    |   movel(pose_trans(ref_frame,p[0.137265, 0.127229, -0.000125, -0.013708, 3.141563, 0.000000]),accel_mss,speed_ms,0,0.001)
    |   movel(pose_trans(ref_frame,p[0.137004, 0.127246, -0.000125, -0.013708, 3.141563, 0.000000]),accel_mss,speed_ms,0,0.001)
    |   movel(pose_trans(ref_frame,p[0.136743, 0.127266, -0.000125, -0.013708, 3.141563, 0.000000]),accel_mss,speed_ms,0,0.001)
    |   movel(pose_trans(ref_frame,p[0.136691, 0.127279, -0.000125, -0.013708, 3.141563, -0.000000]),accel_mss,speed_ms,0,0.001)
    |   movel(pose_trans(ref_frame,p[0.136647, 0.127310, -0.000125, -0.013708, 3.141563, -0.000000]),accel_mss,speed_ms,0,0.001)
    |   movel(pose_trans(ref_frame,p[0.136567, 0.127429, -0.000125, -0.013708, 3.141563, -0.000000]),accel_mss,speed_ms,0,0.001)
    |   movel(pose_trans(ref_frame,p[0.136537, 0.127569, -0.000125, -0.013708, 3.141563, -0.000000]),accel_mss,speed_ms,0,0.001)
    |   movel(pose_trans(ref_frame,p[0.136528, 0.128292, -0.000125, -0.013708, 3.141563, -0.000000]),accel_mss,speed_ms,0,0.001)
    |   movel(pose_trans(ref_frame,p[0.136524, 0.129016, -0.000125, -0.013708, 3.141563, -0.000000]),accel_mss,speed_ms,0,0.001)
    |   movel(pose_trans(ref_frame,p[0.136527, 0.129739, -0.000125, -0.013708, 3.141563, 0.000000]),accel_mss,speed_ms,0,0.001)
    |   movel(pose_trans(ref_frame,p[0.136535, 0.130463, -0.000125, -0.013708, 3.141563, 0.000000]),accel_mss,speed_ms,0,0.001)
    |   movel(pose_trans(ref_frame,p[0.136564, 0.130603, -0.000125, -0.013708, 3.141563, 0.000000]),accel_mss,speed_ms,0,0.001)
    |   movel(pose_trans(ref_frame,p[0.136644, 0.130721, -0.000125, -0.013708, 3.141563, 0.000000]),accel_mss,speed_ms,0,0.001)
    |   movel(pose_trans(ref_frame,p[0.136735, 0.130785, -0.000125, -0.013708, 3.141563, 0.000000]),accel_mss,speed_ms,0,0.001)
    |   movel(pose_trans(ref_frame,p[0.136842, 0.130814, -0.000125, -0.013708, 3.141563, -0.000000]),accel_mss,speed_ms,0,0.001)
    |   movel(pose_trans(ref_frame,p[0.137118, 0.130836, -0.000125, -0.013708, 3.141563, 0.000000]),accel_mss,speed_ms,0,0.001)
    |   movel(pose_trans(ref_frame,p[0.137394, 0.130848, -0.000125, -0.013708, 3.141563, 0.000000]),accel_mss,speed_ms,0,0.001)
    |   movel(pose_trans(ref_frame,p[0.137672, 0.130852, -0.000125, -0.013708, 3.141563, -0.000000]),accel_mss,speed_ms,0,0.001)
    |   movel(pose_trans(ref_frame,p[0.137949, 0.130847, -0.000125, -0.013708, 3.141563, -0.000000]),accel_mss,speed_ms,0,0.001)
    |   movel(pose_trans(ref_frame,p[0.138052, 0.130824, -0.000125, -0.013708, 3.141563, 0.000000]),accel_mss,speed_ms,0,0.001)
    |   movel(pose_trans(ref_frame,p[0.138139, 0.130764, -0.000125, -0.013708, 3.141563, -0.000000]),accel_mss,speed_ms,0,0.001)
    |   movel(pose_trans(ref_frame,p[0.138160, 0.130734, -0.000125, -0.013708, 3.141563, 0.000000]),accel_mss,speed_ms,0,0.001)
    |   movel(pose_trans(ref_frame,p[0.138170, 0.130699, -0.000125, -0.013708, 3.141563, 0.000000]),accel_mss,speed_ms,0,0.001)
    |   movel(pose_trans(ref_frame,p[0.138184, 0.130572, -0.000125, -0.013708, 3.141563, 0.000000]),accel_mss,speed_ms,0,0.001)
    |   movel(pose_trans(ref_frame,p[0.138196, 0.130446, -0.000125, -0.013708, 3.141563, 0.000000]),accel_mss,speed_ms,0,0.001)
    |   movel(pose_trans(ref_frame,p[0.138208, 0.130292, -0.000125, -0.013708, 3.141563, 0.000000]),accel_mss,speed_ms,0,0.001)
    |   movel(pose_trans(ref_frame,p[0.138216, 0.130139, -0.000125, -0.013708, 3.141563, -0.000000]),accel_mss,speed_ms,0,0.001)
    |   movel(pose_trans(ref_frame,p[0.138221, 0.129964, -0.000125, -0.013708, 3.141563, 0.000000]),accel_mss,speed_ms,0,0.001)
    |   movel(pose_trans(ref_frame,p[0.138224, 0.129790, -0.000125, -0.013708, 3.141563, 0.000000]),accel_mss,speed_ms,0,0.001)
    |   movel(pose_trans(ref_frame,p[0.138229, 0.128894, -0.000125, -0.013708, 3.141563, -0.000000]),accel_mss,speed_ms,0,0.001)
    |   movel(pose_trans(ref_frame,p[0.139247, 0.128889, -0.000125, -0.013708, 3.141563, 0.000000]),accel_mss,speed_ms,0,0.001)
    |   movel(pose_trans(ref_frame,p[0.139445, 0.128890, -0.000125, -0.013708, 3.141563, 0.000000]),accel_mss,speed_ms,0,0.001)
    |   movel(pose_trans(ref_frame,p[0.139643, 0.128894, -0.000125, -0.013708, 3.141563, -0.000000]),accel_mss,speed_ms,0,0.001)
    |   movel(pose_trans(ref_frame,p[0.139818, 0.128901, -0.000125, -0.013708, 3.141563, 0.000000]),accel_mss,speed_ms,0,0.001)
    |   movel(pose_trans(ref_frame,p[0.139992, 0.128912, -0.000125, -0.013708, 3.141563, -0.000000]),accel_mss,speed_ms,0,0.001)
    |   movel(pose_trans(ref_frame,p[0.140137, 0.128924, -0.000125, -0.013708, 3.141563, 0.000000]),accel_mss,speed_ms,0,0.001)
    |   movel(pose_trans(ref_frame,p[0.140281, 0.128939, -0.000125, -0.013708, 3.141563, -0.000000]),accel_mss,speed_ms,0,0.001)
    |   movel(pose_trans(ref_frame,p[0.140321, 0.128950, -0.000125, -0.013708, 3.141563, 0.000000]),accel_mss,speed_ms,0,0.001)
    |   movel(pose_trans(ref_frame,p[0.140355, 0.128974, -0.000125, -0.013708, 3.141563, -0.000000]),accel_mss,speed_ms,0,0.001)
    |   movel(pose_trans(ref_frame,p[0.140380, 0.129009, -0.000125, -0.013708, 3.141563, 0.000000]),accel_mss,speed_ms,0,0.001)
    |   movel(pose_trans(ref_frame,p[0.140391, 0.129049, -0.000125, -0.013708, 3.141563, 0.000000]),accel_mss,speed_ms,0,0.001)
    |   movel(pose_trans(ref_frame,p[0.140406, 0.129193, -0.000125, -0.013708, 3.141563, 0.000000]),accel_mss,speed_ms,0,0.001)
    |   movel(pose_trans(ref_frame,p[0.140418, 0.129337, -0.000125, -0.013708, 3.141563, -0.000000]),accel_mss,speed_ms,0,0.001)
    |   movel(pose_trans(ref_frame,p[0.140429, 0.129512, -0.000125, -0.013708, 3.141563, 0.000000]),accel_mss,speed_ms,0,0.001)
    |   movel(pose_trans(ref_frame,p[0.140436, 0.129686, -0.000125, -0.013708, 3.141563, 0.000000]),accel_mss,speed_ms,0,0.001)
    |   movel(pose_trans(ref_frame,p[0.140440, 0.129885, -0.000125, -0.013708, 3.141563, 0.000000]),accel_mss,speed_ms,0,0.001)
    |   movel(pose_trans(ref_frame,p[0.140441, 0.130083, -0.000125, -0.013708, 3.141563, -0.000000]),accel_mss,speed_ms,0,0.001)
    |   movel(pose_trans(ref_frame,p[0.140435, 0.131101, -0.000125, -0.013708, 3.141563, 0.000000]),accel_mss,speed_ms,0,0.001)
    |   movel(pose_trans(ref_frame,p[0.139540, 0.131106, -0.000125, -0.013708, 3.141563, -0.000000]),accel_mss,speed_ms,0,0.001)
    |   movel(pose_trans(ref_frame,p[0.139365, 0.131109, -0.000125, -0.013708, 3.141563, 0.000000]),accel_mss,speed_ms,0,0.001)
    |   movel(pose_trans(ref_frame,p[0.139191, 0.131115, -0.000125, -0.013708, 3.141563, 0.000000]),accel_mss,speed_ms,0,0.001)
    |   movel(pose_trans(ref_frame,p[0.139036, 0.131123, -0.000125, -0.013708, 3.141563, 0.000000]),accel_mss,speed_ms,0,0.001)
    |   movel(pose_trans(ref_frame,p[0.138882, 0.131136, -0.000125, -0.013708, 3.141563, -0.000000]),accel_mss,speed_ms,0,0.001)
    |   movel(pose_trans(ref_frame,p[0.138755, 0.131149, -0.000125, -0.013708, 3.141563, -0.000000]),accel_mss,speed_ms,0,0.001)
    |   movel(pose_trans(ref_frame,p[0.138628, 0.131164, -0.000125, -0.013708, 3.141563, 0.000000]),accel_mss,speed_ms,0,0.001)
    |   movel(pose_trans(ref_frame,p[0.138590, 0.131175, -0.000125, -0.013708, 3.141563, 0.000000]),accel_mss,speed_ms,0,0.001)
    |   movel(pose_trans(ref_frame,p[0.138558, 0.131198, -0.000125, -0.013708, 3.141563, -0.000000]),accel_mss,speed_ms,0,0.001)
    |   movel(pose_trans(ref_frame,p[0.138500, 0.131284, -0.000125, -0.013708, 3.141563, -0.000000]),accel_mss,speed_ms,0,0.001)
    |   movel(pose_trans(ref_frame,p[0.138478, 0.131386, -0.000125, -0.013708, 3.141563, 0.000000]),accel_mss,speed_ms,0,0.001)
    |   movel(pose_trans(ref_frame,p[0.138476, 0.131664, -0.000125, -0.013708, 3.141563, 0.000000]),accel_mss,speed_ms,0,0.001)
    |   movel(pose_trans(ref_frame,p[0.138482, 0.131941, -0.000125, -0.013708, 3.141563, 0.000000]),accel_mss,speed_ms,0,0.001)
    |   movel(pose_trans(ref_frame,p[0.138497, 0.132218, -0.000125, -0.013708, 3.141563, -0.000000]),accel_mss,speed_ms,0,0.001)
    |   movel(pose_trans(ref_frame,p[0.138520, 0.132493, -0.000125, -0.013708, 3.141563, 0.000000]),accel_mss,speed_ms,0,0.001)
    |   movel(pose_trans(ref_frame,p[0.138550, 0.132601, -0.000125, -0.013708, 3.141563, -0.000000]),accel_mss,speed_ms,0,0.001)
    |   movel(pose_trans(ref_frame,p[0.138614, 0.132691, -0.000125, -0.013708, 3.141563, 0.000000]),accel_mss,speed_ms,0,0.001)
    |   movel(pose_trans(ref_frame,p[0.138656, 0.132723, -0.000125, -0.013708, 3.141563, -0.000000]),accel_mss,speed_ms,0,0.001)
    |   movel(pose_trans(ref_frame,p[0.138705, 0.132741, -0.000125, -0.013708, 3.141563, 0.000000]),accel_mss,speed_ms,0,0.001)
    |   movel(pose_trans(ref_frame,p[0.138816, 0.132762, -0.000125, -0.013708, 3.141563, 0.000000]),accel_mss,speed_ms,0,0.001)
    |   movel(pose_trans(ref_frame,p[0.138928, 0.132780, -0.000125, -0.013708, 3.141563, -0.000000]),accel_mss,speed_ms,0,0.001)
    |   movel(pose_trans(ref_frame,p[0.139065, 0.132795, -0.000125, -0.013708, 3.141563, -0.000000]),accel_mss,speed_ms,0,0.001)
    |   movel(pose_trans(ref_frame,p[0.139202, 0.132806, -0.000125, -0.013708, 3.141563, -0.000000]),accel_mss,speed_ms,0,0.001)
    |   movel(pose_trans(ref_frame,p[0.139352, 0.132811, -0.000125, -0.013708, 3.141563, 0.000000]),accel_mss,speed_ms,0,0.001)
    |   movel(pose_trans(ref_frame,p[0.139502, 0.132812, -0.000125, -0.013708, 3.141563, 0.000000]),accel_mss,speed_ms,0,0.001)
    |   movel(pose_trans(ref_frame,p[0.139651, 0.132812, -0.000125, -0.013708, 3.141563, 0.000000]),accel_mss,speed_ms,0,0.001)
    |   movel(pose_trans(ref_frame,p[0.139800, 0.132816, -0.000125, -0.013708, 3.141563, -0.000000]),accel_mss,speed_ms,0,0.001)
    |   movel(pose_trans(ref_frame,p[0.139934, 0.132823, -0.000125, -0.013708, 3.141563, 0.000000]),accel_mss,speed_ms,0,0.001)
    |   movel(pose_trans(ref_frame,p[0.140066, 0.132834, -0.000125, -0.013708, 3.141563, -0.000000]),accel_mss,speed_ms,0,0.001)
    |   movel(pose_trans(ref_frame,p[0.140175, 0.132846, -0.000125, -0.013708, 3.141563, 0.000000]),accel_mss,speed_ms,0,0.001)
    |   movel(pose_trans(ref_frame,p[0.140283, 0.132861, -0.000125, -0.013708, 3.141563, -0.000000]),accel_mss,speed_ms,0,0.001)
    |   movel(pose_trans(ref_frame,p[0.140322, 0.132873, -0.000125, -0.013708, 3.141563, 0.000000]),accel_mss,speed_ms,0,0.001)
    |   movel(pose_trans(ref_frame,p[0.140354, 0.132897, -0.000125, -0.013708, 3.141563, 0.000000]),accel_mss,speed_ms,0,0.001)
    |   movel(pose_trans(ref_frame,p[0.140379, 0.132931, -0.000125, -0.013708, 3.141563, -0.000000]),accel_mss,speed_ms,0,0.001)
    |   movel(pose_trans(ref_frame,p[0.140391, 0.132972, -0.000125, -0.013708, 3.141563, 0.000000]),accel_mss,speed_ms,0,0.001)
    |   movel(pose_trans(ref_frame,p[0.140405, 0.133116, -0.000125, -0.013708, 3.141563, -0.000000]),accel_mss,speed_ms,0,0.001)
    |   movel(pose_trans(ref_frame,p[0.140417, 0.133260, -0.000125, -0.013708, 3.141563, -0.000000]),accel_mss,speed_ms,0,0.001)
    |   movel(pose_trans(ref_frame,p[0.140429, 0.133435, -0.000125, -0.013708, 3.141563, -0.000000]),accel_mss,speed_ms,0,0.001)
    |   movel(pose_trans(ref_frame,p[0.140436, 0.133609, -0.000125, -0.013708, 3.141563, -0.000000]),accel_mss,speed_ms,0,0.001)
    |   movel(pose_trans(ref_frame,p[0.140440, 0.133808, -0.000125, -0.013708, 3.141563, 0.000000]),accel_mss,speed_ms,0,0.001)
    |   movel(pose_trans(ref_frame,p[0.140441, 0.134006, -0.000125, -0.013708, 3.141563, -0.000000]),accel_mss,speed_ms,0,0.001)
    |   movel(pose_trans(ref_frame,p[0.140435, 0.135024, -0.000125, -0.013708, 3.141563, 0.000000]),accel_mss,speed_ms,0,0.001)
    |   movel(pose_trans(ref_frame,p[0.139540, 0.135029, -0.000125, -0.013708, 3.141563, 0.000000]),accel_mss,speed_ms,0,0.001)
    |   movel(pose_trans(ref_frame,p[0.139365, 0.135032, -0.000125, -0.013708, 3.141563, 0.000000]),accel_mss,speed_ms,0,0.001)
    |   movel(pose_trans(ref_frame,p[0.139191, 0.135037, -0.000125, -0.013708, 3.141563, -0.000000]),accel_mss,speed_ms,0,0.001)
    |   movel(pose_trans(ref_frame,p[0.139037, 0.135045, -0.000125, -0.013708, 3.141563, -0.000000]),accel_mss,speed_ms,0,0.001)
    |   movel(pose_trans(ref_frame,p[0.138884, 0.135057, -0.000125, -0.013708, 3.141563, -0.000000]),accel_mss,speed_ms,0,0.001)
    |   movel(pose_trans(ref_frame,p[0.138757, 0.135069, -0.000125, -0.013708, 3.141563, 0.000000]),accel_mss,speed_ms,0,0.001)
    |   movel(pose_trans(ref_frame,p[0.138630, 0.135083, -0.000125, -0.013708, 3.141563, -0.000000]),accel_mss,speed_ms,0,0.001)
    |   movel(pose_trans(ref_frame,p[0.138595, 0.135093, -0.000125, -0.013708, 3.141563, 0.000000]),accel_mss,speed_ms,0,0.001)
    |   movel(pose_trans(ref_frame,p[0.138564, 0.135115, -0.000125, -0.013708, 3.141563, 0.000000]),accel_mss,speed_ms,0,0.001)
    |   movel(pose_trans(ref_frame,p[0.138543, 0.135145, -0.000125, -0.013708, 3.141563, 0.000000]),accel_mss,speed_ms,0,0.001)
    |   movel(pose_trans(ref_frame,p[0.138533, 0.135181, -0.000125, -0.013708, 3.141563, 0.000000]),accel_mss,speed_ms,0,0.001)
    |   movel(pose_trans(ref_frame,p[0.138519, 0.135307, -0.000125, -0.013708, 3.141563, 0.000000]),accel_mss,speed_ms,0,0.001)
    |   movel(pose_trans(ref_frame,p[0.138506, 0.135434, -0.000125, -0.013708, 3.141563, 0.000000]),accel_mss,speed_ms,0,0.001)
    |   movel(pose_trans(ref_frame,p[0.138495, 0.135588, -0.000125, -0.013708, 3.141563, 0.000000]),accel_mss,speed_ms,0,0.001)
    |   movel(pose_trans(ref_frame,p[0.138487, 0.135741, -0.000125, -0.013708, 3.141563, 0.000000]),accel_mss,speed_ms,0,0.001)
    |   movel(pose_trans(ref_frame,p[0.138481, 0.135916, -0.000125, -0.013708, 3.141563, 0.000000]),accel_mss,speed_ms,0,0.001)
    |   movel(pose_trans(ref_frame,p[0.138479, 0.136090, -0.000125, -0.013708, 3.141563, 0.000000]),accel_mss,speed_ms,0,0.001)
    |   movel(pose_trans(ref_frame,p[0.138473, 0.136986, -0.000125, -0.013708, 3.141563, -0.000000]),accel_mss,speed_ms,0,0.001)
    |   movel(pose_trans(ref_frame,p[0.137441, 0.136976, -0.000125, -0.013708, 3.141563, 0.000000]),accel_mss,speed_ms,0,0.001)
    |   movel(pose_trans(ref_frame,p[0.137240, 0.136973, -0.000125, -0.013708, 3.141563, 0.000000]),accel_mss,speed_ms,0,0.001)
    |   movel(pose_trans(ref_frame,p[0.137039, 0.136967, -0.000125, -0.013708, 3.141563, 0.000000]),accel_mss,speed_ms,0,0.001)
    |   movel(pose_trans(ref_frame,p[0.136864, 0.136959, -0.000125, -0.013708, 3.141563, 0.000000]),accel_mss,speed_ms,0,0.001)
    |   movel(pose_trans(ref_frame,p[0.136689, 0.136947, -0.000125, -0.013708, 3.141563, 0.000000]),accel_mss,speed_ms,0,0.001)
    |   movel(pose_trans(ref_frame,p[0.136542, 0.136935, -0.000125, -0.013708, 3.141563, 0.000000]),accel_mss,speed_ms,0,0.001)
    |   movel(pose_trans(ref_frame,p[0.136396, 0.136921, -0.000125, -0.013708, 3.141563, 0.000000]),accel_mss,speed_ms,0,0.001)
    |   movel(pose_trans(ref_frame,p[0.136361, 0.136911, -0.000125, -0.013708, 3.141563, 0.000000]),accel_mss,speed_ms,0,0.001)
    |   movel(pose_trans(ref_frame,p[0.136331, 0.136890, -0.000125, -0.013708, 3.141563, 0.000000]),accel_mss,speed_ms,0,0.001)
    |   movel(pose_trans(ref_frame,p[0.136311, 0.136862, -0.000125, -0.013708, 3.141563, -0.000000]),accel_mss,speed_ms,0,0.001)
    |   movel(pose_trans(ref_frame,p[0.136301, 0.136828, -0.000125, -0.013708, 3.141563, -0.000000]),accel_mss,speed_ms,0,0.001)
    |   movel(pose_trans(ref_frame,p[0.136289, 0.136720, -0.000125, -0.013708, 3.141563, -0.000000]),accel_mss,speed_ms,0,0.001)
    |   movel(pose_trans(ref_frame,p[0.136279, 0.136612, -0.000125, -0.013708, 3.141563, -0.000000]),accel_mss,speed_ms,0,0.001)
    |   movel(pose_trans(ref_frame,p[0.136270, 0.136481, -0.000125, -0.013708, 3.141563, -0.000000]),accel_mss,speed_ms,0,0.001)
    |   movel(pose_trans(ref_frame,p[0.136265, 0.136350, -0.000125, -0.013708, 3.141563, -0.000000]),accel_mss,speed_ms,0,0.001)
    |   movel(pose_trans(ref_frame,p[0.136262, 0.136201, -0.000125, -0.013708, 3.141563, -0.000000]),accel_mss,speed_ms,0,0.001)
    |   movel(pose_trans(ref_frame,p[0.136262, 0.136053, -0.000125, -0.013708, 3.141563, -0.000000]),accel_mss,speed_ms,0,0.001)
    |   movel(pose_trans(ref_frame,p[0.136261, 0.135902, -0.000125, -0.013708, 3.141563, -0.000000]),accel_mss,speed_ms,0,0.001)
    |   movel(pose_trans(ref_frame,p[0.136255, 0.135752, -0.000125, -0.013708, 3.141563, 0.000000]),accel_mss,speed_ms,0,0.001)
    |   movel(pose_trans(ref_frame,p[0.136244, 0.135614, -0.000125, -0.013708, 3.141563, -0.000000]),accel_mss,speed_ms,0,0.001)
    |   movel(pose_trans(ref_frame,p[0.136227, 0.135476, -0.000125, -0.013708, 3.141563, 0.000000]),accel_mss,speed_ms,0,0.001)
    |   movel(pose_trans(ref_frame,p[0.136209, 0.135364, -0.000125, -0.013708, 3.141563, 0.000000]),accel_mss,speed_ms,0,0.001)
    |   movel(pose_trans(ref_frame,p[0.136186, 0.135252, -0.000125, -0.013708, 3.141563, 0.000000]),accel_mss,speed_ms,0,0.001)
    |   movel(pose_trans(ref_frame,p[0.136167, 0.135201, -0.000125, -0.013708, 3.141563, -0.000000]),accel_mss,speed_ms,0,0.001)
    |   movel(pose_trans(ref_frame,p[0.136134, 0.135157, -0.000125, -0.013708, 3.141563, -0.000000]),accel_mss,speed_ms,0,0.001)
    |   movel(pose_trans(ref_frame,p[0.136043, 0.135094, -0.000125, -0.013708, 3.141563, 0.000000]),accel_mss,speed_ms,0,0.001)
    |   movel(pose_trans(ref_frame,p[0.135937, 0.135065, -0.000125, -0.013708, 3.141563, -0.000000]),accel_mss,speed_ms,0,0.001)
    |   movel(pose_trans(ref_frame,p[0.135661, 0.135044, -0.000125, -0.013708, 3.141563, -0.000000]),accel_mss,speed_ms,0,0.001)
    |   movel(pose_trans(ref_frame,p[0.135384, 0.135032, -0.000125, -0.013708, 3.141563, -0.000000]),accel_mss,speed_ms,0,0.001)
    |   movel(pose_trans(ref_frame,p[0.135107, 0.135029, -0.000125, -0.013708, 3.141563, 0.000000]),accel_mss,speed_ms,0,0.001)
    |   movel(pose_trans(ref_frame,p[0.134830, 0.135034, -0.000125, -0.013708, 3.141563, 0.000000]),accel_mss,speed_ms,0,0.001)
    |   movel(pose_trans(ref_frame,p[0.134727, 0.135057, -0.000125, -0.013708, 3.141563, -0.000000]),accel_mss,speed_ms,0,0.001)
    |   movel(pose_trans(ref_frame,p[0.134641, 0.135116, -0.000125, -0.013708, 3.141563, 0.000000]),accel_mss,speed_ms,0,0.001)
    |   movel(pose_trans(ref_frame,p[0.134619, 0.135146, -0.000125, -0.013708, 3.141563, -0.000000]),accel_mss,speed_ms,0,0.001)
    |   movel(pose_trans(ref_frame,p[0.134609, 0.135181, -0.000125, -0.013708, 3.141563, -0.000000]),accel_mss,speed_ms,0,0.001)
    |   movel(pose_trans(ref_frame,p[0.134595, 0.135309, -0.000125, -0.013708, 3.141563, 0.000000]),accel_mss,speed_ms,0,0.001)
    |   movel(pose_trans(ref_frame,p[0.134583, 0.135437, -0.000125, -0.013708, 3.141563, 0.000000]),accel_mss,speed_ms,0,0.001)
    |   movel(pose_trans(ref_frame,p[0.134571, 0.135591, -0.000125, -0.013708, 3.141563, 0.000000]),accel_mss,speed_ms,0,0.001)
    |   movel(pose_trans(ref_frame,p[0.134563, 0.135746, -0.000125, -0.013708, 3.141563, -0.000000]),accel_mss,speed_ms,0,0.001)
    |   movel(pose_trans(ref_frame,p[0.134557, 0.135921, -0.000125, -0.013708, 3.141563, 0.000000]),accel_mss,speed_ms,0,0.001)
    |   movel(pose_trans(ref_frame,p[0.134555, 0.136097, -0.000125, -0.013708, 3.141563, -0.000000]),accel_mss,speed_ms,0,0.001)
    |   movel(pose_trans(ref_frame,p[0.134548, 0.136999, -0.000125, -0.013708, 3.141563, 0.000000]),accel_mss,speed_ms,0,0.001)
    |   movel(pose_trans(ref_frame,p[0.133508, 0.136975, -0.000125, -0.013708, 3.141563, 0.000000]),accel_mss,speed_ms,0,0.001)
    |   movel(pose_trans(ref_frame,p[0.133308, 0.136970, -0.000125, -0.013708, 3.141563, -0.000000]),accel_mss,speed_ms,0,0.001)
    |   movel(pose_trans(ref_frame,p[0.133107, 0.136963, -0.000125, -0.013708, 3.141563, 0.000000]),accel_mss,speed_ms,0,0.001)
    |   movel(pose_trans(ref_frame,p[0.132935, 0.136956, -0.000125, -0.013708, 3.141563, 0.000000]),accel_mss,speed_ms,0,0.001)
    |   movel(pose_trans(ref_frame,p[0.132763, 0.136947, -0.000125, -0.013708, 3.141563, -0.000000]),accel_mss,speed_ms,0,0.001)
    |   movel(pose_trans(ref_frame,p[0.132615, 0.136938, -0.000125, -0.013708, 3.141563, -0.000000]),accel_mss,speed_ms,0,0.001)
    |   movel(pose_trans(ref_frame,p[0.132466, 0.136929, -0.000125, -0.013708, 3.141563, 0.000000]),accel_mss,speed_ms,0,0.001)
    |   movel(pose_trans(ref_frame,p[0.132448, 0.136924, -0.000125, -0.013708, 3.141563, -0.000000]),accel_mss,speed_ms,0,0.001)
    |   movel(pose_trans(ref_frame,p[0.132432, 0.136914, -0.000125, -0.013708, 3.141563, -0.000000]),accel_mss,speed_ms,0,0.001)
    |   movel(pose_trans(ref_frame,p[0.132421, 0.136898, -0.000125, -0.013708, 3.141563, 0.000000]),accel_mss,speed_ms,0,0.001)
    |   movel(pose_trans(ref_frame,p[0.132417, 0.136880, -0.000125, -0.013708, 3.141563, -0.000000]),accel_mss,speed_ms,0,0.001)
    |   movel(pose_trans(ref_frame,p[0.132411, 0.136730, -0.000125, -0.013708, 3.141563, -0.000000]),accel_mss,speed_ms,0,0.001)
    |   movel(pose_trans(ref_frame,p[0.132406, 0.136581, -0.000125, -0.013708, 3.141563, 0.000000]),accel_mss,speed_ms,0,0.001)
    |   movel(pose_trans(ref_frame,p[0.132401, 0.136409, -0.000125, -0.013708, 3.141563, -0.000000]),accel_mss,speed_ms,0,0.001)
    |   movel(pose_trans(ref_frame,p[0.132398, 0.136236, -0.000125, -0.013708, 3.141563, 0.000000]),accel_mss,speed_ms,0,0.001)
    |   movel(pose_trans(ref_frame,p[0.132396, 0.136035, -0.000125, -0.013708, 3.141563, -0.000000]),accel_mss,speed_ms,0,0.001)
    |   movel(pose_trans(ref_frame,p[0.132395, 0.135834, -0.000125, -0.013708, 3.141563, -0.000000]),accel_mss,speed_ms,0,0.001)
    |   movel(pose_trans(ref_frame,p[0.132395, 0.134791, -0.000125, -0.013708, 3.141563, 0.000000]),accel_mss,speed_ms,0,0.001)
    |   movel(pose_trans(ref_frame,p[0.133279, 0.134766, -0.000125, -0.013708, 3.141563, 0.000000]),accel_mss,speed_ms,0,0.001)
    |   movel(pose_trans(ref_frame,p[0.133451, 0.134760, -0.000125, -0.013708, 3.141563, 0.000000]),accel_mss,speed_ms,0,0.001)
    |   movel(pose_trans(ref_frame,p[0.133623, 0.134751, -0.000125, -0.013708, 3.141563, 0.000000]),accel_mss,speed_ms,0,0.001)
    |   movel(pose_trans(ref_frame,p[0.133774, 0.134741, -0.000125, -0.013708, 3.141563, 0.000000]),accel_mss,speed_ms,0,0.001)
    |   movel(pose_trans(ref_frame,p[0.133924, 0.134727, -0.000125, -0.013708, 3.141563, 0.000000]),accel_mss,speed_ms,0,0.001)
    |   movel(pose_trans(ref_frame,p[0.134049, 0.134713, -0.000125, -0.013708, 3.141563, 0.000000]),accel_mss,speed_ms,0,0.001)
    |   movel(pose_trans(ref_frame,p[0.134174, 0.134698, -0.000125, -0.013708, 3.141563, 0.000000]),accel_mss,speed_ms,0,0.001)
    |   movel(pose_trans(ref_frame,p[0.134207, 0.134688, -0.000125, -0.013708, 3.141563, -0.000000]),accel_mss,speed_ms,0,0.001)
    |   movel(pose_trans(ref_frame,p[0.134235, 0.134668, -0.000125, -0.013708, 3.141563, 0.000000]),accel_mss,speed_ms,0,0.001)
    |   movel(pose_trans(ref_frame,p[0.134289, 0.134588, -0.000125, -0.013708, 3.141563, -0.000000]),accel_mss,speed_ms,0,0.001)
    |   movel(pose_trans(ref_frame,p[0.134309, 0.134492, -0.000125, -0.013708, 3.141563, -0.000000]),accel_mss,speed_ms,0,0.001)
    |   movel(pose_trans(ref_frame,p[0.134307, 0.134213, -0.000125, -0.013708, 3.141563, 0.000000]),accel_mss,speed_ms,0,0.001)
    |   movel(pose_trans(ref_frame,p[0.134298, 0.133934, -0.000125, -0.013708, 3.141563, 0.000000]),accel_mss,speed_ms,0,0.001)
    |   movel(pose_trans(ref_frame,p[0.134281, 0.133656, -0.000125, -0.013708, 3.141563, 0.000000]),accel_mss,speed_ms,0,0.001)
    |   movel(pose_trans(ref_frame,p[0.134257, 0.133379, -0.000125, -0.013708, 3.141563, -0.000000]),accel_mss,speed_ms,0,0.001)
    |   movel(pose_trans(ref_frame,p[0.134228, 0.133277, -0.000125, -0.013708, 3.141563, -0.000000]),accel_mss,speed_ms,0,0.001)
    |   movel(pose_trans(ref_frame,p[0.134167, 0.133191, -0.000125, -0.013708, 3.141563, -0.000000]),accel_mss,speed_ms,0,0.001)
    |   movel(pose_trans(ref_frame,p[0.134055, 0.133115, -0.000125, -0.013708, 3.141563, 0.000000]),accel_mss,speed_ms,0,0.001)
    |   movel(pose_trans(ref_frame,p[0.133921, 0.133086, -0.000125, -0.013708, 3.141563, -0.000000]),accel_mss,speed_ms,0,0.001)
    |   movel(pose_trans(ref_frame,p[0.133197, 0.133076, -0.000125, -0.013708, 3.141563, -0.000000]),accel_mss,speed_ms,0,0.001)
    |   movel(pose_trans(ref_frame,p[0.132473, 0.133070, -0.000125, -0.013708, 3.141563, 0.000000]),accel_mss,speed_ms,0,0.001)
    |   movel(pose_trans(ref_frame,p[0.131748, 0.133070, -0.000125, -0.013708, 3.141563, 0.000000]),accel_mss,speed_ms,0,0.001)
    |   movel(pose_trans(ref_frame,p[0.131024, 0.133075, -0.000125, -0.013708, 3.141563, 0.000000]),accel_mss,speed_ms,0,0.001)
    |   movel(pose_trans(ref_frame,p[0.130892, 0.133102, -0.000125, -0.013708, 3.141563, -0.000000]),accel_mss,speed_ms,0,0.001)
    |   movel(pose_trans(ref_frame,p[0.130779, 0.133178, -0.000125, -0.013708, 3.141563, 0.000000]),accel_mss,speed_ms,0,0.001)
    |   movel(pose_trans(ref_frame,p[0.130750, 0.133221, -0.000125, -0.013708, 3.141563, 0.000000]),accel_mss,speed_ms,0,0.001)
    |   movel(pose_trans(ref_frame,p[0.130736, 0.133271, -0.000125, -0.013708, 3.141563, 0.000000]),accel_mss,speed_ms,0,0.001)
    |   movel(pose_trans(ref_frame,p[0.130718, 0.133527, -0.000125, -0.013708, 3.141563, 0.000000]),accel_mss,speed_ms,0,0.001)
    |   movel(pose_trans(ref_frame,p[0.130701, 0.133784, -0.000125, -0.013708, 3.141563, 0.000000]),accel_mss,speed_ms,0,0.001)
    |   movel(pose_trans(ref_frame,p[0.130685, 0.134087, -0.000125, -0.013708, 3.141563, -0.000000]),accel_mss,speed_ms,0,0.001)
    |   movel(pose_trans(ref_frame,p[0.130674, 0.134391, -0.000125, -0.013708, 3.141563, -0.000000]),accel_mss,speed_ms,0,0.001)
    |   movel(pose_trans(ref_frame,p[0.130666, 0.134741, -0.000125, -0.013708, 3.141563, 0.000000]),accel_mss,speed_ms,0,0.001)
    |   movel(pose_trans(ref_frame,p[0.130662, 0.135091, -0.000125, -0.013708, 3.141563, 0.000000]),accel_mss,speed_ms,0,0.001)
    |   movel(pose_trans(ref_frame,p[0.130658, 0.135438, -0.000125, -0.013708, 3.141563, -0.000000]),accel_mss,speed_ms,0,0.001)
    |   movel(pose_trans(ref_frame,p[0.130652, 0.135786, -0.000125, -0.013708, 3.141563, 0.000000]),accel_mss,speed_ms,0,0.001)
    |   movel(pose_trans(ref_frame,p[0.130643, 0.136081, -0.000125, -0.013708, 3.141563, -0.000000]),accel_mss,speed_ms,0,0.001)
    |   movel(pose_trans(ref_frame,p[0.130630, 0.136377, -0.000125, -0.013708, 3.141563, -0.000000]),accel_mss,speed_ms,0,0.001)
    |   movel(pose_trans(ref_frame,p[0.130616, 0.136631, -0.000125, -0.013708, 3.141563, -0.000000]),accel_mss,speed_ms,0,0.001)
    |   movel(pose_trans(ref_frame,p[0.130602, 0.136885, -0.000125, -0.013708, 3.141563, 0.000000]),accel_mss,speed_ms,0,0.001)
    |   movel(pose_trans(ref_frame,p[0.130591, 0.136914, -0.000125, -0.013708, 3.141563, 0.000000]),accel_mss,speed_ms,0,0.001)
    |   movel(pose_trans(ref_frame,p[0.130568, 0.136933, -0.000125, -0.013708, 3.141563, 0.000000]),accel_mss,speed_ms,0,0.001)
    |   movel(pose_trans(ref_frame,p[0.130533, 0.136944, -0.000125, -0.013708, 3.141563, 0.000000]),accel_mss,speed_ms,0,0.001)
    |   movel(pose_trans(ref_frame,p[0.130496, 0.136948, -0.000125, -0.013708, 3.141563, -0.000000]),accel_mss,speed_ms,0,0.001)
    |   movel(pose_trans(ref_frame,p[0.115124, 0.136974, -0.000125, -0.013708, 3.141563, -0.000000]),accel_mss,speed_ms,0,0.001)
    |   movel(pose_trans(ref_frame,p[0.106662, 0.136988, -0.000125, -0.013708, 3.141563, 0.000000]),accel_mss,speed_ms,0,0.001)
    |   movel(pose_trans(ref_frame,p[0.098199, 0.136999, -0.000125, -0.013708, 3.141563, 0.000000]),accel_mss,speed_ms,0,0.001)
    |   movel(pose_trans(ref_frame,p[0.088155, 0.137011, -0.000125, -0.013708, 3.141563, 0.000000]),accel_mss,speed_ms,0,0.001)
    |   movel(pose_trans(ref_frame,p[0.078111, 0.137022, -0.000125, -0.013708, 3.141563, -0.000000]),accel_mss,speed_ms,0,0.001)
    |   movel(pose_trans(ref_frame,p[0.025738, 0.137075, -0.000125, -0.013708, 3.141563, 0.000000]),accel_mss,speed_ms,0,0.001)
    |   movel(pose_trans(ref_frame,p[0.025735, 0.135241, -0.000125, -0.013708, 3.141563, -0.000000]),accel_mss,speed_ms,0,0.001)
    |   movel(pose_trans(ref_frame,p[0.025732, 0.134884, -0.000125, -0.013708, 3.141563, -0.000000]),accel_mss,speed_ms,0,0.001)
    |   movel(pose_trans(ref_frame,p[0.025724, 0.134528, -0.000125, -0.013708, 3.141563, 0.000000]),accel_mss,speed_ms,0,0.001)
    |   movel(pose_trans(ref_frame,p[0.025713, 0.134218, -0.000125, -0.013708, 3.141563, 0.000000]),accel_mss,speed_ms,0,0.001)
    |   movel(pose_trans(ref_frame,p[0.025695, 0.133908, -0.000125, -0.013708, 3.141563, -0.000000]),accel_mss,speed_ms,0,0.001)
    |   movel(pose_trans(ref_frame,p[0.025676, 0.133648, -0.000125, -0.013708, 3.141563, 0.000000]),accel_mss,speed_ms,0,0.001)
    |   movel(pose_trans(ref_frame,p[0.025655, 0.133388, -0.000125, -0.013708, 3.141563, 0.000000]),accel_mss,speed_ms,0,0.001)
    |   movel(pose_trans(ref_frame,p[0.025639, 0.133329, -0.000125, -0.013708, 3.141563, 0.000000]),accel_mss,speed_ms,0,0.001)
    |   movel(pose_trans(ref_frame,p[0.025604, 0.133278, -0.000125, -0.013708, 3.141563, -0.000000]),accel_mss,speed_ms,0,0.001)
    |   movel(pose_trans(ref_frame,p[0.025480, 0.133195, -0.000125, -0.013708, 3.141563, -0.000000]),accel_mss,speed_ms,0,0.001)
    |   movel(pose_trans(ref_frame,p[0.025335, 0.133165, -0.000125, -0.013708, 3.141563, -0.000000]),accel_mss,speed_ms,0,0.001)
    |   movel(pose_trans(ref_frame,p[0.024616, 0.133157, -0.000125, -0.013708, 3.141563, -0.000000]),accel_mss,speed_ms,0,0.001)
    |   movel(pose_trans(ref_frame,p[0.023897, 0.133156, -0.000125, -0.013708, 3.141563, -0.000000]),accel_mss,speed_ms,0,0.001)
    |   movel(pose_trans(ref_frame,p[0.023178, 0.133161, -0.000125, -0.013708, 3.141563, 0.000000]),accel_mss,speed_ms,0,0.001)
    |   movel(pose_trans(ref_frame,p[0.022459, 0.133172, -0.000125, -0.013708, 3.141563, 0.000000]),accel_mss,speed_ms,0,0.001)
    |   movel(pose_trans(ref_frame,p[0.022313, 0.133204, -0.000125, -0.013708, 3.141563, -0.000000]),accel_mss,speed_ms,0,0.001)
    |   movel(pose_trans(ref_frame,p[0.022189, 0.133287, -0.000125, -0.013708, 3.141563, -0.000000]),accel_mss,speed_ms,0,0.001)
    |   movel(pose_trans(ref_frame,p[0.022117, 0.133391, -0.000125, -0.013708, 3.141563, 0.000000]),accel_mss,speed_ms,0,0.001)
    |   movel(pose_trans(ref_frame,p[0.022084, 0.133512, -0.000125, -0.013708, 3.141563, 0.000000]),accel_mss,speed_ms,0,0.001)
    |   movel(pose_trans(ref_frame,p[0.022070, 0.133748, -0.000125, -0.013708, 3.141563, 0.000000]),accel_mss,speed_ms,0,0.001)
    |   movel(pose_trans(ref_frame,p[0.022071, 0.133983, -0.000125, -0.013708, 3.141563, -0.000000]),accel_mss,speed_ms,0,0.001)
    |   movel(pose_trans(ref_frame,p[0.022087, 0.134220, -0.000125, -0.013708, 3.141563, 0.000000]),accel_mss,speed_ms,0,0.001)
    |   movel(pose_trans(ref_frame,p[0.022119, 0.134454, -0.000125, -0.013708, 3.141563, 0.000000]),accel_mss,speed_ms,0,0.001)
    |   movel(pose_trans(ref_frame,p[0.022160, 0.134581, -0.000125, -0.013708, 3.141563, -0.000000]),accel_mss,speed_ms,0,0.001)
    |   movel(pose_trans(ref_frame,p[0.022239, 0.134690, -0.000125, -0.013708, 3.141563, 0.000000]),accel_mss,speed_ms,0,0.001)
    |   movel(pose_trans(ref_frame,p[0.022291, 0.134729, -0.000125, -0.013708, 3.141563, 0.000000]),accel_mss,speed_ms,0,0.001)
    |   movel(pose_trans(ref_frame,p[0.022350, 0.134754, -0.000125, -0.013708, 3.141563, 0.000000]),accel_mss,speed_ms,0,0.001)
    |   movel(pose_trans(ref_frame,p[0.022471, 0.134783, -0.000125, -0.013708, 3.141563, -0.000000]),accel_mss,speed_ms,0,0.001)
    |   movel(pose_trans(ref_frame,p[0.022593, 0.134807, -0.000125, -0.013708, 3.141563, 0.000000]),accel_mss,speed_ms,0,0.001)
    |   movel(pose_trans(ref_frame,p[0.022741, 0.134829, -0.000125, -0.013708, 3.141563, 0.000000]),accel_mss,speed_ms,0,0.001)
    |   movel(pose_trans(ref_frame,p[0.022891, 0.134845, -0.000125, -0.013708, 3.141563, 0.000000]),accel_mss,speed_ms,0,0.001)
    |   movel(pose_trans(ref_frame,p[0.023052, 0.134855, -0.000125, -0.013708, 3.141563, 0.000000]),accel_mss,speed_ms,0,0.001)
    |   movel(pose_trans(ref_frame,p[0.023213, 0.134859, -0.000125, -0.013708, 3.141563, 0.000000]),accel_mss,speed_ms,0,0.001)
    |   movel(pose_trans(ref_frame,p[0.024024, 0.134865, -0.000125, -0.013708, 3.141563, 0.000000]),accel_mss,speed_ms,0,0.001)
    |   movel(pose_trans(ref_frame,p[0.024029, 0.135970, -0.000125, -0.013708, 3.141563, 0.000000]),accel_mss,speed_ms,0,0.001)
    |   movel(pose_trans(ref_frame,p[0.024034, 0.137075, -0.000125, -0.013708, 3.141563, -0.000000]),accel_mss,speed_ms,0,0.001)
    |   movel(pose_trans(ref_frame,p[0.022932, 0.137075, -0.000125, -0.013708, 3.141563, 0.000000]),accel_mss,speed_ms,0,0.001)
    |   movel(pose_trans(ref_frame,p[0.021829, 0.137075, -0.000125, -0.013708, 3.141563, 0.000000]),accel_mss,speed_ms,0,0.001)
    |   movel(pose_trans(ref_frame,p[0.021877, 0.136331, -0.000125, -0.013708, 3.141563, 0.000000]),accel_mss,speed_ms,0,0.001)
    |   movel(pose_trans(ref_frame,p[0.021890, 0.135997, -0.000125, -0.013708, 3.141563, -0.000000]),accel_mss,speed_ms,0,0.001)
    |   movel(pose_trans(ref_frame,p[0.021886, 0.135664, -0.000125, -0.013708, 3.141563, -0.000000]),accel_mss,speed_ms,0,0.001)
    |   movel(pose_trans(ref_frame,p[0.021855, 0.135492, -0.000125, -0.013708, 3.141563, 0.000000]),accel_mss,speed_ms,0,0.001)
    |   movel(pose_trans(ref_frame,p[0.021777, 0.135336, -0.000125, -0.013708, 3.141563, -0.000000]),accel_mss,speed_ms,0,0.001)
    |   movel(pose_trans(ref_frame,p[0.021666, 0.135228, -0.000125, -0.013708, 3.141563, -0.000000]),accel_mss,speed_ms,0,0.001)
    |   movel(pose_trans(ref_frame,p[0.021524, 0.135169, -0.000125, -0.013708, 3.141563, -0.000000]),accel_mss,speed_ms,0,0.001)
    |   movel(pose_trans(ref_frame,p[0.021277, 0.135130, -0.000125, -0.013708, 3.141563, -0.000000]),accel_mss,speed_ms,0,0.001)
    |   movel(pose_trans(ref_frame,p[0.021026, 0.135115, -0.000125, -0.013708, 3.141563, -0.000000]),accel_mss,speed_ms,0,0.001)
    |   movel(pose_trans(ref_frame,p[0.020896, 0.135115, -0.000125, -0.013708, 3.141563, 0.000000]),accel_mss,speed_ms,0,0.001)
    |   movel(pose_trans(ref_frame,p[0.020766, 0.135121, -0.000125, -0.013708, 3.141563, 0.000000]),accel_mss,speed_ms,0,0.001)
    |   movel(pose_trans(ref_frame,p[0.020646, 0.135130, -0.000125, -0.013708, 3.141563, 0.000000]),accel_mss,speed_ms,0,0.001)
    |   movel(pose_trans(ref_frame,p[0.020527, 0.135145, -0.000125, -0.013708, 3.141563, 0.000000]),accel_mss,speed_ms,0,0.001)
    |   movel(pose_trans(ref_frame,p[0.020430, 0.135161, -0.000125, -0.013708, 3.141563, 0.000000]),accel_mss,speed_ms,0,0.001)
    |   movel(pose_trans(ref_frame,p[0.020333, 0.135181, -0.000125, -0.013708, 3.141563, 0.000000]),accel_mss,speed_ms,0,0.001)
    |   movel(pose_trans(ref_frame,p[0.020288, 0.135199, -0.000125, -0.013708, 3.141563, 0.000000]),accel_mss,speed_ms,0,0.001)
    |   movel(pose_trans(ref_frame,p[0.020249, 0.135228, -0.000125, -0.013708, 3.141563, 0.000000]),accel_mss,speed_ms,0,0.001)
    |   movel(pose_trans(ref_frame,p[0.020218, 0.135270, -0.000125, -0.013708, 3.141563, 0.000000]),accel_mss,speed_ms,0,0.001)
    |   movel(pose_trans(ref_frame,p[0.020202, 0.135319, -0.000125, -0.013708, 3.141563, 0.000000]),accel_mss,speed_ms,0,0.001)
    |   movel(pose_trans(ref_frame,p[0.020183, 0.135442, -0.000125, -0.013708, 3.141563, 0.000000]),accel_mss,speed_ms,0,0.001)
    |   movel(pose_trans(ref_frame,p[0.020167, 0.135567, -0.000125, -0.013708, 3.141563, 0.000000]),accel_mss,speed_ms,0,0.001)
    |   movel(pose_trans(ref_frame,p[0.020153, 0.135719, -0.000125, -0.013708, 3.141563, -0.000000]),accel_mss,speed_ms,0,0.001)
    |   movel(pose_trans(ref_frame,p[0.020145, 0.135872, -0.000125, -0.013708, 3.141563, -0.000000]),accel_mss,speed_ms,0,0.001)
    |   movel(pose_trans(ref_frame,p[0.020141, 0.136041, -0.000125, -0.013708, 3.141563, -0.000000]),accel_mss,speed_ms,0,0.001)
    |   movel(pose_trans(ref_frame,p[0.020141, 0.136210, -0.000125, -0.013708, 3.141563, -0.000000]),accel_mss,speed_ms,0,0.001)
    |   movel(pose_trans(ref_frame,p[0.020155, 0.137072, -0.000125, -0.013708, 3.141563, 0.000000]),accel_mss,speed_ms,0,0.001)
    |   movel(pose_trans(ref_frame,p[0.019067, 0.137076, -0.000125, -0.013708, 3.141563, 0.000000]),accel_mss,speed_ms,0,0.001)
    |   movel(pose_trans(ref_frame,p[0.017979, 0.137081, -0.000125, -0.013708, 3.141563, 0.000000]),accel_mss,speed_ms,0,0.001)
    |   movel(pose_trans(ref_frame,p[0.017974, 0.136223, -0.000125, -0.013708, 3.141563, -0.000000]),accel_mss,speed_ms,0,0.001)
    |   movel(pose_trans(ref_frame,p[0.017971, 0.136054, -0.000125, -0.013708, 3.141563, -0.000000]),accel_mss,speed_ms,0,0.001)
    |   movel(pose_trans(ref_frame,p[0.017963, 0.135886, -0.000125, -0.013708, 3.141563, 0.000000]),accel_mss,speed_ms,0,0.001)
    |   movel(pose_trans(ref_frame,p[0.017951, 0.135733, -0.000125, -0.013708, 3.141563, 0.000000]),accel_mss,speed_ms,0,0.001)
    |   movel(pose_trans(ref_frame,p[0.017934, 0.135581, -0.000125, -0.013708, 3.141563, -0.000000]),accel_mss,speed_ms,0,0.001)
    |   movel(pose_trans(ref_frame,p[0.017916, 0.135457, -0.000125, -0.013708, 3.141563, 0.000000]),accel_mss,speed_ms,0,0.001)
    |   movel(pose_trans(ref_frame,p[0.017894, 0.135334, -0.000125, -0.013708, 3.141563, 0.000000]),accel_mss,speed_ms,0,0.001)
    |   movel(pose_trans(ref_frame,p[0.017877, 0.135285, -0.000125, -0.013708, 3.141563, 0.000000]),accel_mss,speed_ms,0,0.001)
    |   movel(pose_trans(ref_frame,p[0.017846, 0.135243, -0.000125, -0.013708, 3.141563, -0.000000]),accel_mss,speed_ms,0,0.001)
    |   movel(pose_trans(ref_frame,p[0.017804, 0.135212, -0.000125, -0.013708, 3.141563, -0.000000]),accel_mss,speed_ms,0,0.001)
    |   movel(pose_trans(ref_frame,p[0.017755, 0.135194, -0.000125, -0.013708, 3.141563, 0.000000]),accel_mss,speed_ms,0,0.001)
    |   movel(pose_trans(ref_frame,p[0.017631, 0.135173, -0.000125, -0.013708, 3.141563, -0.000000]),accel_mss,speed_ms,0,0.001)
    |   movel(pose_trans(ref_frame,p[0.017507, 0.135155, -0.000125, -0.013708, 3.141563, 0.000000]),accel_mss,speed_ms,0,0.001)
    |   movel(pose_trans(ref_frame,p[0.017355, 0.135138, -0.000125, -0.013708, 3.141563, 0.000000]),accel_mss,speed_ms,0,0.001)
    |   movel(pose_trans(ref_frame,p[0.017203, 0.135126, -0.000125, -0.013708, 3.141563, -0.000000]),accel_mss,speed_ms,0,0.001)
    |   movel(pose_trans(ref_frame,p[0.017034, 0.135118, -0.000125, -0.013708, 3.141563, 0.000000]),accel_mss,speed_ms,0,0.001)
    |   movel(pose_trans(ref_frame,p[0.016865, 0.135115, -0.000125, -0.013708, 3.141563, -0.000000]),accel_mss,speed_ms,0,0.001)
    |   movel(pose_trans(ref_frame,p[0.016008, 0.135109, -0.000125, -0.013708, 3.141563, -0.000000]),accel_mss,speed_ms,0,0.001)
    |   movel(pose_trans(ref_frame,p[0.016011, 0.134006, -0.000125, -0.013708, 3.141563, -0.000000]),accel_mss,speed_ms,0,0) # end trace
    |   speed_ms    = 1.000
    |   movel(pose_trans(ref_frame,p[0.016011, 0.134006, 0.005000, -0.013708, 3.141563, -0.000000]),accel_mss,speed_ms,0,0.001)
    |   movel(pose_trans(ref_frame,p[0.000000, 0.000000, 0.005000, -0.013708, 3.141563, 0.000000]),accel_mss,speed_ms,0,0.001)
    |   movel(pose_trans(ref_frame,p[0.000000, 0.000000, 0.055000, -0.013708, 3.141563, -0.000000]),accel_mss,speed_ms,0,0.001)
    |   # End of main program
    | end
    | 
    | output_middle()
  Script file /programs/usbdisk/output_RSettings.script
    | def output_RSettings():
    |   # Global parameters:
    |   global speed_ms    = 0.250
    |   global speed_rads  = 0.750
    |   global accel_mss   = 1.200
    |   global accel_radss = 1.200
    |   global blend_radius_m = 0.001
    |   global ref_frame = p[0,0,0,0,0,0]
    | 
    |   #
    |   # TO REMOVE HEADER:
    |   # Go to "Program" -> "Post-Processor Editor"
    |   # Select "Universal Robots"
    |   # Set "INCLUDE_HEADER" to "False"
    |   #
    |   #--------------------------
    |   # Add any default subprograms here
    |   # For example, to drive a gripper as a program call:
    |   # def Gripper_Open():
    |   #   ...
    |   # end
    |   #
    |   # Example to drive a spray gun:
    |   def SprayOn(value):
    |     # use the value as an output:
    |     DO_SPRAY = 5
    |     if value == 0:
    |       set_standard_digital_out(DO_SPRAY, False)
    |     else:
    |       set_standard_digital_out(DO_SPRAY, True)
    |     end
    |   end
    | 
    |   # Example to drive an extruder:
    |   def Extruder(value):
    |     # use the value as an output:
    |     if value < 0:
    |       # stop extruder
    |     else:
    |       # start extruder
    |     end
    |   end
    | 
    |   # Example to move an external axis
    |   def MoveAxis(value):
    |     # use the value as an output:
    |     DO_AXIS_1 = 1
    |     DI_AXIS_1 = 1
    |     if value <= 0:
    |       set_standard_digital_out(DO_AXIS_1, False)
    | 
    |       # Wait for digital input to change state
    |       #while (get_standard_digital_in(DI_AXIS_1) != False):
    |       #  sync()
    |       #end
    |     else:
    |       set_standard_digital_out(DO_AXIS_1, True)
    | 
    |       # Wait for digital input to change state
    |       #while (get_standard_digital_in(DI_AXIS_1) != True):
    |       #  sync()
    |       #end
    |     end
    |   end
    |   #--------------------------
    | 
    | 
    |   # Main program:
    |   # Program generated by RoboDK v5.7.4 for UR10e on 08/01/2025 21:21:43
    |   # Using nominal kinematics.
    |   blend_radius_m = 0.001
    |   speed_ms    = 1.000
    |   ref_frame = p[0.326125, 0.122767, 0.009000, 0.000000, 0.000000, -0.008727]
    |   set_tcp(p[0.000000, 0.000000, 0.252000, 0.000000, 0.000000, 0.000000])
    |   # Show Tool
    |   movej([0.854487, -1.303262, -2.473446, -0.935678, 1.570796, 2.425275],accel_radss,speed_rads,0,0)
    |   movel(pose_trans(ref_frame,p[0.078892, 0.078720, 0.005000, -0.013708, 3.141563, 0.000000]),accel_mss,speed_ms,0,0) # end trace
    |   speed_ms    = 0.002
    |   movel(pose_trans(ref_frame,p[0.078892, 0.078720, -0.000125, -0.013708, 3.141563, -0.000000]),accel_mss,speed_ms,0,0) # end trace
    |   speed_ms    = 0.007
    |   movel(pose_trans(ref_frame,p[0.079868, 0.078932, -0.000125, -0.013708, 3.141563, 0.000000]),accel_mss,speed_ms,0,0.001)
    |   movel(pose_trans(ref_frame,p[0.080833, 0.079163, -0.000125, -0.013708, 3.141563, 0.000000]),accel_mss,speed_ms,0,0.001)
    |   movel(pose_trans(ref_frame,p[0.081602, 0.079416, -0.000125, -0.013708, 3.141563, -0.000000]),accel_mss,speed_ms,0,0.001)
    |   movel(pose_trans(ref_frame,p[0.082359, 0.079687, -0.000125, -0.013708, 3.141563, -0.000000]),accel_mss,speed_ms,0,0.001)
    |   movel(pose_trans(ref_frame,p[0.086688, 0.081714, -0.000125, -0.013708, 3.141563, 0.000000]),accel_mss,speed_ms,0,0.001)
    |   movel(pose_trans(ref_frame,p[0.090570, 0.084347, -0.000125, -0.013708, 3.141563, 0.000000]),accel_mss,speed_ms,0,0.001)
    |   movel(pose_trans(ref_frame,p[0.091420, 0.085053, -0.000125, -0.013708, 3.141563, 0.000000]),accel_mss,speed_ms,0,0.001)
    |   movel(pose_trans(ref_frame,p[0.092243, 0.085789, -0.000125, -0.013708, 3.141563, -0.000000]),accel_mss,speed_ms,0,0.001)
    |   movel(pose_trans(ref_frame,p[0.092902, 0.086419, -0.000125, -0.013708, 3.141563, 0.000000]),accel_mss,speed_ms,0,0.001)
    |   movel(pose_trans(ref_frame,p[0.093542, 0.087070, -0.000125, -0.013708, 3.141563, 0.000000]),accel_mss,speed_ms,0,0.001)
    |   movel(pose_trans(ref_frame,p[0.093889, 0.087440, -0.000125, -0.013708, 3.141563, 0.000000]),accel_mss,speed_ms,0,0.001)
    |   movel(pose_trans(ref_frame,p[0.094230, 0.087815, -0.000125, -0.013708, 3.141563, 0.000000]),accel_mss,speed_ms,0,0.001)
    |   movel(pose_trans(ref_frame,p[0.094772, 0.088440, -0.000125, -0.013708, 3.141563, 0.000000]),accel_mss,speed_ms,0,0.001)
    |   movel(pose_trans(ref_frame,p[0.095297, 0.089081, -0.000125, -0.013708, 3.141563, -0.000000]),accel_mss,speed_ms,0,0.001)
    |   movel(pose_trans(ref_frame,p[0.095678, 0.089569, -0.000125, -0.013708, 3.141563, 0.000000]),accel_mss,speed_ms,0,0.001)
    |   movel(pose_trans(ref_frame,p[0.096049, 0.090066, -0.000125, -0.013708, 3.141563, 0.000000]),accel_mss,speed_ms,0,0.001)
    |   movel(pose_trans(ref_frame,p[0.097201, 0.091759, -0.000125, -0.013708, 3.141563, -0.000000]),accel_mss,speed_ms,0,0.001)
    |   movel(pose_trans(ref_frame,p[0.098242, 0.093541, -0.000125, -0.013708, 3.141563, -0.000000]),accel_mss,speed_ms,0,0.001)
    |   movel(pose_trans(ref_frame,p[0.098866, 0.094765, -0.000125, -0.013708, 3.141563, 0.000000]),accel_mss,speed_ms,0,0.001)
    |   movel(pose_trans(ref_frame,p[0.099437, 0.096026, -0.000125, -0.013708, 3.141563, 0.000000]),accel_mss,speed_ms,0,0.001)
    |   movel(pose_trans(ref_frame,p[0.100019, 0.097672, -0.000125, -0.013708, 3.141563, 0.000000]),accel_mss,speed_ms,0,0.001)
    |   movel(pose_trans(ref_frame,p[0.100523, 0.099369, -0.000125, -0.013708, 3.141563, 0.000000]),accel_mss,speed_ms,0,0) # end trace
    |   speed_ms    = 1.000
    |   movel(pose_trans(ref_frame,p[0.100523, 0.099369, 0.005000, -0.013708, 3.141563, 0.000000]),accel_mss,speed_ms,0,0.001)
    |   movel(pose_trans(ref_frame,p[0.087112, 0.102660, 0.005000, -0.013708, 3.141563, -0.000000]),accel_mss,speed_ms,0,0) # end trace
    |   speed_ms    = 0.002
    |   movel(pose_trans(ref_frame,p[0.087112, 0.102660, -0.000125, -0.013708, 3.141563, -0.000000]),accel_mss,speed_ms,0,0) # end trace
    |   speed_ms    = 0.007
    |   movel(pose_trans(ref_frame,p[0.087463, 0.102752, -0.000125, -0.013708, 3.141563, -0.000000]),accel_mss,speed_ms,0,0.001)
    |   movel(pose_trans(ref_frame,p[0.087821, 0.102816, -0.000125, -0.013708, 3.141563, 0.000000]),accel_mss,speed_ms,0,0.001)
    |   movel(pose_trans(ref_frame,p[0.088167, 0.102847, -0.000125, -0.013708, 3.141563, 0.000000]),accel_mss,speed_ms,0,0.001)
    |   movel(pose_trans(ref_frame,p[0.088514, 0.102847, -0.000125, -0.013708, 3.141563, 0.000000]),accel_mss,speed_ms,0,0.001)
    |   movel(pose_trans(ref_frame,p[0.088877, 0.102814, -0.000125, -0.013708, 3.141563, 0.000000]),accel_mss,speed_ms,0,0.001)
    |   movel(pose_trans(ref_frame,p[0.089235, 0.102751, -0.000125, -0.013708, 3.141563, 0.000000]),accel_mss,speed_ms,0,0.001)
    |   movel(pose_trans(ref_frame,p[0.089634, 0.102650, -0.000125, -0.013708, 3.141563, 0.000000]),accel_mss,speed_ms,0,0.001)
    |   movel(pose_trans(ref_frame,p[0.090026, 0.102526, -0.000125, -0.013708, 3.141563, -0.000000]),accel_mss,speed_ms,0,0.001)
    |   movel(pose_trans(ref_frame,p[0.090266, 0.102437, -0.000125, -0.013708, 3.141563, -0.000000]),accel_mss,speed_ms,0,0.001)
    |   movel(pose_trans(ref_frame,p[0.090502, 0.102340, -0.000125, -0.013708, 3.141563, -0.000000]),accel_mss,speed_ms,0,0.001)
    |   movel(pose_trans(ref_frame,p[0.090671, 0.102259, -0.000125, -0.013708, 3.141563, 0.000000]),accel_mss,speed_ms,0,0.001)
    |   movel(pose_trans(ref_frame,p[0.090831, 0.102163, -0.000125, -0.013708, 3.141563, 0.000000]),accel_mss,speed_ms,0,0.001)
    |   movel(pose_trans(ref_frame,p[0.090992, 0.102049, -0.000125, -0.013708, 3.141563, 0.000000]),accel_mss,speed_ms,0,0.001)
    |   movel(pose_trans(ref_frame,p[0.091143, 0.101922, -0.000125, -0.013708, 3.141563, 0.000000]),accel_mss,speed_ms,0,0.001)
    |   movel(pose_trans(ref_frame,p[0.091360, 0.101720, -0.000125, -0.013708, 3.141563, -0.000000]),accel_mss,speed_ms,0,0.001)
    |   movel(pose_trans(ref_frame,p[0.091572, 0.101513, -0.000125, -0.013708, 3.141563, 0.000000]),accel_mss,speed_ms,0,0.001)
    |   movel(pose_trans(ref_frame,p[0.091779, 0.101301, -0.000125, -0.013708, 3.141563, 0.000000]),accel_mss,speed_ms,0,0.001)
    |   movel(pose_trans(ref_frame,p[0.091981, 0.101085, -0.000125, -0.013708, 3.141563, 0.000000]),accel_mss,speed_ms,0,0.001)
    |   movel(pose_trans(ref_frame,p[0.092104, 0.100938, -0.000125, -0.013708, 3.141563, 0.000000]),accel_mss,speed_ms,0,0.001)
    |   movel(pose_trans(ref_frame,p[0.092216, 0.100781, -0.000125, -0.013708, 3.141563, 0.000000]),accel_mss,speed_ms,0,0.001)
    |   movel(pose_trans(ref_frame,p[0.092307, 0.100629, -0.000125, -0.013708, 3.141563, 0.000000]),accel_mss,speed_ms,0,0.001)
    |   movel(pose_trans(ref_frame,p[0.092383, 0.100468, -0.000125, -0.013708, 3.141563, 0.000000]),accel_mss,speed_ms,0,0.001)
    |   movel(pose_trans(ref_frame,p[0.092470, 0.100248, -0.000125, -0.013708, 3.141563, -0.000000]),accel_mss,speed_ms,0,0.001)
    |   movel(pose_trans(ref_frame,p[0.092549, 0.100024, -0.000125, -0.013708, 3.141563, 0.000000]),accel_mss,speed_ms,0,0.001)
    |   movel(pose_trans(ref_frame,p[0.092669, 0.099587, -0.000125, -0.013708, 3.141563, -0.000000]),accel_mss,speed_ms,0,0.001)
    |   movel(pose_trans(ref_frame,p[0.092743, 0.099139, -0.000125, -0.013708, 3.141563, 0.000000]),accel_mss,speed_ms,0,0.001)
    |   movel(pose_trans(ref_frame,p[0.092785, 0.098610, -0.000125, -0.013708, 3.141563, 0.000000]),accel_mss,speed_ms,0,0.001)
    |   movel(pose_trans(ref_frame,p[0.092793, 0.098080, -0.000125, -0.013708, 3.141563, -0.000000]),accel_mss,speed_ms,0,0.001)
    |   movel(pose_trans(ref_frame,p[0.092765, 0.097519, -0.000125, -0.013708, 3.141563, 0.000000]),accel_mss,speed_ms,0,0.001)
    |   movel(pose_trans(ref_frame,p[0.092703, 0.096961, -0.000125, -0.013708, 3.141563, 0.000000]),accel_mss,speed_ms,0,0.001)
    |   movel(pose_trans(ref_frame,p[0.092608, 0.096423, -0.000125, -0.013708, 3.141563, -0.000000]),accel_mss,speed_ms,0,0.001)
    |   movel(pose_trans(ref_frame,p[0.092476, 0.095893, -0.000125, -0.013708, 3.141563, -0.000000]),accel_mss,speed_ms,0,0.001)
    |   movel(pose_trans(ref_frame,p[0.092409, 0.095667, -0.000125, -0.013708, 3.141563, 0.000000]),accel_mss,speed_ms,0,0.001)
    |   movel(pose_trans(ref_frame,p[0.092337, 0.095443, -0.000125, -0.013708, 3.141563, 0.000000]),accel_mss,speed_ms,0,0.001)
    |   movel(pose_trans(ref_frame,p[0.092262, 0.095233, -0.000125, -0.013708, 3.141563, 0.000000]),accel_mss,speed_ms,0,0.001)
    |   movel(pose_trans(ref_frame,p[0.092182, 0.095026, -0.000125, -0.013708, 3.141563, 0.000000]),accel_mss,speed_ms,0,0.001)
    |   movel(pose_trans(ref_frame,p[0.092110, 0.094854, -0.000125, -0.013708, 3.141563, -0.000000]),accel_mss,speed_ms,0,0.001)
    |   movel(pose_trans(ref_frame,p[0.092033, 0.094685, -0.000125, -0.013708, 3.141563, -0.000000]),accel_mss,speed_ms,0,0.001)
    |   movel(pose_trans(ref_frame,p[0.091986, 0.094604, -0.000125, -0.013708, 3.141563, 0.000000]),accel_mss,speed_ms,0,0.001)
    |   movel(pose_trans(ref_frame,p[0.091926, 0.094532, -0.000125, -0.013708, 3.141563, -0.000000]),accel_mss,speed_ms,0,0.001)
    |   movel(pose_trans(ref_frame,p[0.091668, 0.094355, -0.000125, -0.013708, 3.141563, 0.000000]),accel_mss,speed_ms,0,0.001)
    |   movel(pose_trans(ref_frame,p[0.091363, 0.094284, -0.000125, -0.013708, 3.141563, 0.000000]),accel_mss,speed_ms,0,0.001)
    |   movel(pose_trans(ref_frame,p[0.090817, 0.094283, -0.000125, -0.013708, 3.141563, 0.000000]),accel_mss,speed_ms,0,0.001)
    |   movel(pose_trans(ref_frame,p[0.090272, 0.094324, -0.000125, -0.013708, 3.141563, 0.000000]),accel_mss,speed_ms,0,0.001)
    |   movel(pose_trans(ref_frame,p[0.089634, 0.094424, -0.000125, -0.013708, 3.141563, 0.000000]),accel_mss,speed_ms,0,0.001)
    |   movel(pose_trans(ref_frame,p[0.089006, 0.094572, -0.000125, -0.013708, 3.141563, -0.000000]),accel_mss,speed_ms,0,0.001)
    |   movel(pose_trans(ref_frame,p[0.088394, 0.094768, -0.000125, -0.013708, 3.141563, 0.000000]),accel_mss,speed_ms,0,0.001)
    |   movel(pose_trans(ref_frame,p[0.087800, 0.095012, -0.000125, -0.013708, 3.141563, 0.000000]),accel_mss,speed_ms,0,0.001)
    |   movel(pose_trans(ref_frame,p[0.087450, 0.095185, -0.000125, -0.013708, 3.141563, -0.000000]),accel_mss,speed_ms,0,0.001)
    |   movel(pose_trans(ref_frame,p[0.087113, 0.095382, -0.000125, -0.013708, 3.141563, 0.000000]),accel_mss,speed_ms,0,0.001)
    |   movel(pose_trans(ref_frame,p[0.086733, 0.095631, -0.000125, -0.013708, 3.141563, 0.000000]),accel_mss,speed_ms,0,0.001)
    |   movel(pose_trans(ref_frame,p[0.086364, 0.095897, -0.000125, -0.013708, 3.141563, -0.000000]),accel_mss,speed_ms,0,0.001)
    |   movel(pose_trans(ref_frame,p[0.086019, 0.096167, -0.000125, -0.013708, 3.141563, 0.000000]),accel_mss,speed_ms,0,0.001)
    |   movel(pose_trans(ref_frame,p[0.085686, 0.096452, -0.000125, -0.013708, 3.141563, 0.000000]),accel_mss,speed_ms,0,0.001)
    |   movel(pose_trans(ref_frame,p[0.085448, 0.096684, -0.000125, -0.013708, 3.141563, -0.000000]),accel_mss,speed_ms,0,0.001)
    |   movel(pose_trans(ref_frame,p[0.085234, 0.096938, -0.000125, -0.013708, 3.141563, 0.000000]),accel_mss,speed_ms,0,0.001)
    |   movel(pose_trans(ref_frame,p[0.084848, 0.097539, -0.000125, -0.013708, 3.141563, -0.000000]),accel_mss,speed_ms,0,0.001)
    |   movel(pose_trans(ref_frame,p[0.084569, 0.098197, -0.000125, -0.013708, 3.141563, -0.000000]),accel_mss,speed_ms,0,0.001)
    |   movel(pose_trans(ref_frame,p[0.084427, 0.098849, -0.000125, -0.013708, 3.141563, -0.000000]),accel_mss,speed_ms,0,0.001)
    |   movel(pose_trans(ref_frame,p[0.084421, 0.099516, -0.000125, -0.013708, 3.141563, -0.000000]),accel_mss,speed_ms,0,0.001)
    |   movel(pose_trans(ref_frame,p[0.084552, 0.100168, -0.000125, -0.013708, 3.141563, -0.000000]),accel_mss,speed_ms,0,0.001)
    |   movel(pose_trans(ref_frame,p[0.084815, 0.100779, -0.000125, -0.013708, 3.141563, -0.000000]),accel_mss,speed_ms,0,0.001)
    |   movel(pose_trans(ref_frame,p[0.085213, 0.101368, -0.000125, -0.013708, 3.141563, 0.000000]),accel_mss,speed_ms,0,0.001)
    |   movel(pose_trans(ref_frame,p[0.085705, 0.101880, -0.000125, -0.013708, 3.141563, -0.000000]),accel_mss,speed_ms,0,0.001)
    |   movel(pose_trans(ref_frame,p[0.085871, 0.102020, -0.000125, -0.013708, 3.141563, -0.000000]),accel_mss,speed_ms,0,0.001)
    |   movel(pose_trans(ref_frame,p[0.086043, 0.102153, -0.000125, -0.013708, 3.141563, -0.000000]),accel_mss,speed_ms,0,0.001)
    |   movel(pose_trans(ref_frame,p[0.086196, 0.102259, -0.000125, -0.013708, 3.141563, 0.000000]),accel_mss,speed_ms,0,0.001)
    |   movel(pose_trans(ref_frame,p[0.086357, 0.102355, -0.000125, -0.013708, 3.141563, 0.000000]),accel_mss,speed_ms,0,0.001)
    |   movel(pose_trans(ref_frame,p[0.086524, 0.102440, -0.000125, -0.013708, 3.141563, 0.000000]),accel_mss,speed_ms,0,0.001)
    |   movel(pose_trans(ref_frame,p[0.086696, 0.102515, -0.000125, -0.013708, 3.141563, 0.000000]),accel_mss,speed_ms,0,0.001)
    |   movel(pose_trans(ref_frame,p[0.086903, 0.102592, -0.000125, -0.013708, 3.141563, 0.000000]),accel_mss,speed_ms,0,0.001)
    |   movel(pose_trans(ref_frame,p[0.087112, 0.102660, -0.000125, -0.013708, 3.141563, -0.000000]),accel_mss,speed_ms,0,0) # end trace
    |   speed_ms    = 1.000
    |   movel(pose_trans(ref_frame,p[0.087112, 0.102660, 0.005000, -0.013708, 3.141563, -0.000000]),accel_mss,speed_ms,0,0.001)
    |   movel(pose_trans(ref_frame,p[0.094089, 0.085862, 0.005000, -0.013708, 3.141563, 0.000000]),accel_mss,speed_ms,0,0) # end trace
    |   speed_ms    = 0.002
    |   movel(pose_trans(ref_frame,p[0.094089, 0.085862, -0.000125, -0.013708, 3.141563, -0.000000]),accel_mss,speed_ms,0,0) # end trace
    |   speed_ms    = 0.007
    |   movel(pose_trans(ref_frame,p[0.094841, 0.086283, -0.000125, -0.013708, 3.141563, -0.000000]),accel_mss,speed_ms,0,0.001)
    |   movel(pose_trans(ref_frame,p[0.095642, 0.086599, -0.000125, -0.013708, 3.141563, 0.000000]),accel_mss,speed_ms,0,0.001)
    |   movel(pose_trans(ref_frame,p[0.096468, 0.086800, -0.000125, -0.013708, 3.141563, 0.000000]),accel_mss,speed_ms,0,0.001)
    |   movel(pose_trans(ref_frame,p[0.097314, 0.086884, -0.000125, -0.013708, 3.141563, -0.000000]),accel_mss,speed_ms,0,0.001)
    |   movel(pose_trans(ref_frame,p[0.098161, 0.086848, -0.000125, -0.013708, 3.141563, 0.000000]),accel_mss,speed_ms,0,0.001)
    |   movel(pose_trans(ref_frame,p[0.098996, 0.086694, -0.000125, -0.013708, 3.141563, 0.000000]),accel_mss,speed_ms,0,0.001)
    |   movel(pose_trans(ref_frame,p[0.099811, 0.086424, -0.000125, -0.013708, 3.141563, -0.000000]),accel_mss,speed_ms,0,0.001)
    |   movel(pose_trans(ref_frame,p[0.100581, 0.086046, -0.000125, -0.013708, 3.141563, 0.000000]),accel_mss,speed_ms,0,0.001)
    |   movel(pose_trans(ref_frame,p[0.100885, 0.085851, -0.000125, -0.013708, 3.141563, 0.000000]),accel_mss,speed_ms,0,0.001)
    |   movel(pose_trans(ref_frame,p[0.101171, 0.085631, -0.000125, -0.013708, 3.141563, 0.000000]),accel_mss,speed_ms,0,0.001)
    |   movel(pose_trans(ref_frame,p[0.101509, 0.085331, -0.000125, -0.013708, 3.141563, 0.000000]),accel_mss,speed_ms,0,0.001)
    |   movel(pose_trans(ref_frame,p[0.101833, 0.085016, -0.000125, -0.013708, 3.141563, 0.000000]),accel_mss,speed_ms,0,0.001)
    |   movel(pose_trans(ref_frame,p[0.102141, 0.084687, -0.000125, -0.013708, 3.141563, 0.000000]),accel_mss,speed_ms,0,0.001)
    |   movel(pose_trans(ref_frame,p[0.102433, 0.084345, -0.000125, -0.013708, 3.141563, 0.000000]),accel_mss,speed_ms,0,0.001)
    |   movel(pose_trans(ref_frame,p[0.102643, 0.084061, -0.000125, -0.013708, 3.141563, 0.000000]),accel_mss,speed_ms,0,0.001)
    |   movel(pose_trans(ref_frame,p[0.102826, 0.083759, -0.000125, -0.013708, 3.141563, -0.000000]),accel_mss,speed_ms,0,0.001)
    |   movel(pose_trans(ref_frame,p[0.103021, 0.083373, -0.000125, -0.013708, 3.141563, -0.000000]),accel_mss,speed_ms,0,0.001)
    |   movel(pose_trans(ref_frame,p[0.103192, 0.082976, -0.000125, -0.013708, 3.141563, 0.000000]),accel_mss,speed_ms,0,0.001)
    |   movel(pose_trans(ref_frame,p[0.103321, 0.082608, -0.000125, -0.013708, 3.141563, 0.000000]),accel_mss,speed_ms,0,0.001)
    |   movel(pose_trans(ref_frame,p[0.103420, 0.082230, -0.000125, -0.013708, 3.141563, 0.000000]),accel_mss,speed_ms,0,0.001)
    |   movel(pose_trans(ref_frame,p[0.103497, 0.081807, -0.000125, -0.013708, 3.141563, -0.000000]),accel_mss,speed_ms,0,0.001)
    |   movel(pose_trans(ref_frame,p[0.103544, 0.081379, -0.000125, -0.013708, 3.141563, -0.000000]),accel_mss,speed_ms,0,0.001)
    |   movel(pose_trans(ref_frame,p[0.103577, 0.080821, -0.000125, -0.013708, 3.141563, -0.000000]),accel_mss,speed_ms,0,0.001)
    |   movel(pose_trans(ref_frame,p[0.103591, 0.080261, -0.000125, -0.013708, 3.141563, -0.000000]),accel_mss,speed_ms,0,0.001)
    |   movel(pose_trans(ref_frame,p[0.103596, 0.079949, -0.000125, -0.013708, 3.141563, 0.000000]),accel_mss,speed_ms,0,0.001)
    |   movel(pose_trans(ref_frame,p[0.103603, 0.079636, -0.000125, -0.013708, 3.141563, 0.000000]),accel_mss,speed_ms,0,0.001)
    |   movel(pose_trans(ref_frame,p[0.103613, 0.079367, -0.000125, -0.013708, 3.141563, -0.000000]),accel_mss,speed_ms,0,0.001)
    |   movel(pose_trans(ref_frame,p[0.103627, 0.079097, -0.000125, -0.013708, 3.141563, 0.000000]),accel_mss,speed_ms,0,0.001)
    |   movel(pose_trans(ref_frame,p[0.103641, 0.078868, -0.000125, -0.013708, 3.141563, -0.000000]),accel_mss,speed_ms,0,0.001)
    |   movel(pose_trans(ref_frame,p[0.103656, 0.078638, -0.000125, -0.013708, 3.141563, -0.000000]),accel_mss,speed_ms,0,0.001)
    |   movel(pose_trans(ref_frame,p[0.103666, 0.078599, -0.000125, -0.013708, 3.141563, 0.000000]),accel_mss,speed_ms,0,0.001)
    |   movel(pose_trans(ref_frame,p[0.103689, 0.078565, -0.000125, -0.013708, 3.141563, 0.000000]),accel_mss,speed_ms,0,0.001)
    |   movel(pose_trans(ref_frame,p[0.103723, 0.078542, -0.000125, -0.013708, 3.141563, 0.000000]),accel_mss,speed_ms,0,0.001)
    |   movel(pose_trans(ref_frame,p[0.103763, 0.078532, -0.000125, -0.013708, 3.141563, 0.000000]),accel_mss,speed_ms,0,0.001)
    |   movel(pose_trans(ref_frame,p[0.104018, 0.078519, -0.000125, -0.013708, 3.141563, -0.000000]),accel_mss,speed_ms,0,0.001)
    |   movel(pose_trans(ref_frame,p[0.104272, 0.078508, -0.000125, -0.013708, 3.141563, -0.000000]),accel_mss,speed_ms,0,0.001)
    |   movel(pose_trans(ref_frame,p[0.104570, 0.078498, -0.000125, -0.013708, 3.141563, -0.000000]),accel_mss,speed_ms,0,0.001)
    |   movel(pose_trans(ref_frame,p[0.104868, 0.078491, -0.000125, -0.013708, 3.141563, 0.000000]),accel_mss,speed_ms,0,0.001)
    |   movel(pose_trans(ref_frame,p[0.105213, 0.078487, -0.000125, -0.013708, 3.141563, -0.000000]),accel_mss,speed_ms,0,0.001)
    |   movel(pose_trans(ref_frame,p[0.105559, 0.078486, -0.000125, -0.013708, 3.141563, -0.000000]),accel_mss,speed_ms,0,0.001)
    |   movel(pose_trans(ref_frame,p[0.105906, 0.078485, -0.000125, -0.013708, 3.141563, -0.000000]),accel_mss,speed_ms,0,0.001)
    |   movel(pose_trans(ref_frame,p[0.106253, 0.078479, -0.000125, -0.013708, 3.141563, -0.000000]),accel_mss,speed_ms,0,0.001)
    |   movel(pose_trans(ref_frame,p[0.106555, 0.078469, -0.000125, -0.013708, 3.141563, 0.000000]),accel_mss,speed_ms,0,0.001)
    |   movel(pose_trans(ref_frame,p[0.106857, 0.078453, -0.000125, -0.013708, 3.141563, 0.000000]),accel_mss,speed_ms,0,0.001)
    |   movel(pose_trans(ref_frame,p[0.107110, 0.078436, -0.000125, -0.013708, 3.141563, -0.000000]),accel_mss,speed_ms,0,0.001)
    |   movel(pose_trans(ref_frame,p[0.107363, 0.078417, -0.000125, -0.013708, 3.141563, 0.000000]),accel_mss,speed_ms,0,0.001)
    |   movel(pose_trans(ref_frame,p[0.107419, 0.078402, -0.000125, -0.013708, 3.141563, 0.000000]),accel_mss,speed_ms,0,0.001)
    |   movel(pose_trans(ref_frame,p[0.107467, 0.078369, -0.000125, -0.013708, 3.141563, 0.000000]),accel_mss,speed_ms,0,0.001)
    |   movel(pose_trans(ref_frame,p[0.107550, 0.078247, -0.000125, -0.013708, 3.141563, -0.000000]),accel_mss,speed_ms,0,0.001)
    |   movel(pose_trans(ref_frame,p[0.107580, 0.078103, -0.000125, -0.013708, 3.141563, 0.000000]),accel_mss,speed_ms,0,0.001)
    |   movel(pose_trans(ref_frame,p[0.107584, 0.077925, -0.000125, -0.013708, 3.141563, -0.000000]),accel_mss,speed_ms,0,0.001)
    |   movel(pose_trans(ref_frame,p[0.107587, 0.077748, -0.000125, -0.013708, 3.141563, 0.000000]),accel_mss,speed_ms,0,0.001)
    |   movel(pose_trans(ref_frame,p[0.107591, 0.077466, -0.000125, -0.013708, 3.141563, 0.000000]),accel_mss,speed_ms,0,0.001)
    |   movel(pose_trans(ref_frame,p[0.107594, 0.077183, -0.000125, -0.013708, 3.141563, 0.000000]),accel_mss,speed_ms,0,0.001)
    |   movel(pose_trans(ref_frame,p[0.107597, 0.076879, -0.000125, -0.013708, 3.141563, 0.000000]),accel_mss,speed_ms,0,0.001)
    |   movel(pose_trans(ref_frame,p[0.107599, 0.076575, -0.000125, -0.013708, 3.141563, 0.000000]),accel_mss,speed_ms,0,0.001)
    |   movel(pose_trans(ref_frame,p[0.107600, 0.076211, -0.000125, -0.013708, 3.141563, 0.000000]),accel_mss,speed_ms,0,0.001)
    |   movel(pose_trans(ref_frame,p[0.107599, 0.075847, -0.000125, -0.013708, 3.141563, 0.000000]),accel_mss,speed_ms,0,0.001)
    |   movel(pose_trans(ref_frame,p[0.107594, 0.075047, -0.000125, -0.013708, 3.141563, 0.000000]),accel_mss,speed_ms,0,0.001)
    |   movel(pose_trans(ref_frame,p[0.107565, 0.074904, -0.000125, -0.013708, 3.141563, -0.000000]),accel_mss,speed_ms,0,0.001)
    |   movel(pose_trans(ref_frame,p[0.107483, 0.074782, -0.000125, -0.013708, 3.141563, -0.000000]),accel_mss,speed_ms,0,0.001)
    |   movel(pose_trans(ref_frame,p[0.107343, 0.074689, -0.000125, -0.013708, 3.141563, -0.000000]),accel_mss,speed_ms,0,0.001)
    |   movel(pose_trans(ref_frame,p[0.107178, 0.074656, -0.000125, -0.013708, 3.141563, -0.000000]),accel_mss,speed_ms,0,0.001)
    |   movel(pose_trans(ref_frame,p[0.106570, 0.074655, -0.000125, -0.013708, 3.141563, 0.000000]),accel_mss,speed_ms,0,0.001)
    |   movel(pose_trans(ref_frame,p[0.105872, 0.074655, -0.000125, -0.013708, 3.141563, 0.000000]),accel_mss,speed_ms,0,0.001)
    |   movel(pose_trans(ref_frame,p[0.105247, 0.074654, -0.000125, -0.013708, 3.141563, -0.000000]),accel_mss,speed_ms,0,0.001)
    |   movel(pose_trans(ref_frame,p[0.104230, 0.074653, -0.000125, -0.013708, 3.141563, 0.000000]),accel_mss,speed_ms,0,0.001)
    |   movel(pose_trans(ref_frame,p[0.103267, 0.074653, -0.000125, -0.013708, 3.141563, 0.000000]),accel_mss,speed_ms,0,0.001)
    |   movel(pose_trans(ref_frame,p[0.102412, 0.074652, -0.000125, -0.013708, 3.141563, 0.000000]),accel_mss,speed_ms,0,0.001)
    |   movel(pose_trans(ref_frame,p[0.101678, 0.074651, -0.000125, -0.013708, 3.141563, 0.000000]),accel_mss,speed_ms,0,0.001)
    |   movel(pose_trans(ref_frame,p[0.101407, 0.074651, -0.000125, -0.013708, 3.141563, -0.000000]),accel_mss,speed_ms,0,0.001)
    |   movel(pose_trans(ref_frame,p[0.101075, 0.074651, -0.000125, -0.013708, 3.141563, -0.000000]),accel_mss,speed_ms,0,0.001)
    |   movel(pose_trans(ref_frame,p[0.099984, 0.074652, -0.000125, -0.013708, 3.141563, -0.000000]),accel_mss,speed_ms,0,0.001)
    |   movel(pose_trans(ref_frame,p[0.099535, 0.074653, -0.000125, -0.013708, 3.141563, 0.000000]),accel_mss,speed_ms,0,0.001)
    |   movel(pose_trans(ref_frame,p[0.099054, 0.074653, -0.000125, -0.013708, 3.141563, 0.000000]),accel_mss,speed_ms,0,0.001)
    |   movel(pose_trans(ref_frame,p[0.098648, 0.074653, -0.000125, -0.013708, 3.141563, 0.000000]),accel_mss,speed_ms,0,0.001)
    |   movel(pose_trans(ref_frame,p[0.098254, 0.074653, -0.000125, -0.013708, 3.141563, 0.000000]),accel_mss,speed_ms,0,0.001)
    |   movel(pose_trans(ref_frame,p[0.097920, 0.074654, -0.000125, -0.013708, 3.141563, -0.000000]),accel_mss,speed_ms,0,0.001)
    |   movel(pose_trans(ref_frame,p[0.097614, 0.074654, -0.000125, -0.013708, 3.141563, 0.000000]),accel_mss,speed_ms,0,0.001)
    |   movel(pose_trans(ref_frame,p[0.097253, 0.074654, -0.000125, -0.013708, 3.141563, 0.000000]),accel_mss,speed_ms,0,0.001)
    |   movel(pose_trans(ref_frame,p[0.096960, 0.074654, -0.000125, -0.013708, 3.141563, -0.000000]),accel_mss,speed_ms,0,0.001)
    |   movel(pose_trans(ref_frame,p[0.096532, 0.074655, -0.000125, -0.013708, 3.141563, 0.000000]),accel_mss,speed_ms,0,0.001)
    |   movel(pose_trans(ref_frame,p[0.096178, 0.074655, -0.000125, -0.013708, 3.141563, 0.000000]),accel_mss,speed_ms,0,0.001)
    |   movel(pose_trans(ref_frame,p[0.096013, 0.074688, -0.000125, -0.013708, 3.141563, 0.000000]),accel_mss,speed_ms,0,0.001)
    |   movel(pose_trans(ref_frame,p[0.095874, 0.074782, -0.000125, -0.013708, 3.141563, -0.000000]),accel_mss,speed_ms,0,0.001)
    |   movel(pose_trans(ref_frame,p[0.095792, 0.074903, -0.000125, -0.013708, 3.141563, -0.000000]),accel_mss,speed_ms,0,0.001)
    |   movel(pose_trans(ref_frame,p[0.095762, 0.075047, -0.000125, -0.013708, 3.141563, 0.000000]),accel_mss,speed_ms,0,0.001)
    |   movel(pose_trans(ref_frame,p[0.095759, 0.075277, -0.000125, -0.013708, 3.141563, -0.000000]),accel_mss,speed_ms,0,0.001)
    |   movel(pose_trans(ref_frame,p[0.095758, 0.075508, -0.000125, -0.013708, 3.141563, 0.000000]),accel_mss,speed_ms,0,0.001)
    |   movel(pose_trans(ref_frame,p[0.095758, 0.075703, -0.000125, -0.013708, 3.141563, 0.000000]),accel_mss,speed_ms,0,0.001)
    |   movel(pose_trans(ref_frame,p[0.095755, 0.075898, -0.000125, -0.013708, 3.141563, 0.000000]),accel_mss,speed_ms,0,0.001)
    |   movel(pose_trans(ref_frame,p[0.095755, 0.076237, -0.000125, -0.013708, 3.141563, 0.000000]),accel_mss,speed_ms,0,0.001)
    |   movel(pose_trans(ref_frame,p[0.095755, 0.076575, -0.000125, -0.013708, 3.141563, 0.000000]),accel_mss,speed_ms,0,0.001)
    |   movel(pose_trans(ref_frame,p[0.095757, 0.076868, -0.000125, -0.013708, 3.141563, 0.000000]),accel_mss,speed_ms,0,0.001)
    |   movel(pose_trans(ref_frame,p[0.095759, 0.077162, -0.000125, -0.013708, 3.141563, -0.000000]),accel_mss,speed_ms,0,0.001)
    |   movel(pose_trans(ref_frame,p[0.095763, 0.077415, -0.000125, -0.013708, 3.141563, 0.000000]),accel_mss,speed_ms,0,0.001)
    |   movel(pose_trans(ref_frame,p[0.095766, 0.077667, -0.000125, -0.013708, 3.141563, 0.000000]),accel_mss,speed_ms,0,0.001)
    |   movel(pose_trans(ref_frame,p[0.095773, 0.078102, -0.000125, -0.013708, 3.141563, 0.000000]),accel_mss,speed_ms,0,0.001)
    |   movel(pose_trans(ref_frame,p[0.095805, 0.078247, -0.000125, -0.013708, 3.141563, -0.000000]),accel_mss,speed_ms,0,0.001)
    |   movel(pose_trans(ref_frame,p[0.095887, 0.078369, -0.000125, -0.013708, 3.141563, -0.000000]),accel_mss,speed_ms,0,0.001)
    |   movel(pose_trans(ref_frame,p[0.095935, 0.078403, -0.000125, -0.013708, 3.141563, 0.000000]),accel_mss,speed_ms,0,0.001)
    |   movel(pose_trans(ref_frame,p[0.095991, 0.078417, -0.000125, -0.013708, 3.141563, -0.000000]),accel_mss,speed_ms,0,0.001)
    |   movel(pose_trans(ref_frame,p[0.096244, 0.078437, -0.000125, -0.013708, 3.141563, -0.000000]),accel_mss,speed_ms,0,0.001)
    |   movel(pose_trans(ref_frame,p[0.096497, 0.078453, -0.000125, -0.013708, 3.141563, -0.000000]),accel_mss,speed_ms,0,0.001)
    |   movel(pose_trans(ref_frame,p[0.096799, 0.078469, -0.000125, -0.013708, 3.141563, 0.000000]),accel_mss,speed_ms,0,0.001)
    |   movel(pose_trans(ref_frame,p[0.097101, 0.078479, -0.000125, -0.013708, 3.141563, 0.000000]),accel_mss,speed_ms,0,0.001)
    |   movel(pose_trans(ref_frame,p[0.097448, 0.078485, -0.000125, -0.013708, 3.141563, -0.000000]),accel_mss,speed_ms,0,0.001)
    |   movel(pose_trans(ref_frame,p[0.097795, 0.078486, -0.000125, -0.013708, 3.141563, 0.000000]),accel_mss,speed_ms,0,0.001)
    |   movel(pose_trans(ref_frame,p[0.098141, 0.078488, -0.000125, -0.013708, 3.141563, 0.000000]),accel_mss,speed_ms,0,0.001)
    |   movel(pose_trans(ref_frame,p[0.098487, 0.078492, -0.000125, -0.013708, 3.141563, -0.000000]),accel_mss,speed_ms,0,0.001)
    |   movel(pose_trans(ref_frame,p[0.098786, 0.078500, -0.000125, -0.013708, 3.141563, 0.000000]),accel_mss,speed_ms,0,0.001)
    |   movel(pose_trans(ref_frame,p[0.099085, 0.078512, -0.000125, -0.013708, 3.141563, 0.000000]),accel_mss,speed_ms,0,0.001)
    |   movel(pose_trans(ref_frame,p[0.099339, 0.078525, -0.000125, -0.013708, 3.141563, -0.000000]),accel_mss,speed_ms,0,0.001)
    |   movel(pose_trans(ref_frame,p[0.099593, 0.078540, -0.000125, -0.013708, 3.141563, 0.000000]),accel_mss,speed_ms,0,0.001)
    |   movel(pose_trans(ref_frame,p[0.099638, 0.078551, -0.000125, -0.013708, 3.141563, 0.000000]),accel_mss,speed_ms,0,0.001)
    |   movel(pose_trans(ref_frame,p[0.099677, 0.078577, -0.000125, -0.013708, 3.141563, -0.000000]),accel_mss,speed_ms,0,0.001)
    |   movel(pose_trans(ref_frame,p[0.099753, 0.078692, -0.000125, -0.013708, 3.141563, 0.000000]),accel_mss,speed_ms,0,0.001)
    |   movel(pose_trans(ref_frame,p[0.099778, 0.078828, -0.000125, -0.013708, 3.141563, -0.000000]),accel_mss,speed_ms,0,0.001)
    |   movel(pose_trans(ref_frame,p[0.099766, 0.079401, -0.000125, -0.013708, 3.141563, -0.000000]),accel_mss,speed_ms,0,0.001)
    |   movel(pose_trans(ref_frame,p[0.099746, 0.079974, -0.000125, -0.013708, 3.141563, 0.000000]),accel_mss,speed_ms,0,0.001)
    |   movel(pose_trans(ref_frame,p[0.099718, 0.080526, -0.000125, -0.013708, 3.141563, 0.000000]),accel_mss,speed_ms,0,0.001)
    |   movel(pose_trans(ref_frame,p[0.099678, 0.081077, -0.000125, -0.013708, 3.141563, 0.000000]),accel_mss,speed_ms,0,0.001)
    |   movel(pose_trans(ref_frame,p[0.099636, 0.081338, -0.000125, -0.013708, 3.141563, 0.000000]),accel_mss,speed_ms,0,0.001)
    |   movel(pose_trans(ref_frame,p[0.099555, 0.081590, -0.000125, -0.013708, 3.141563, 0.000000]),accel_mss,speed_ms,0,0.001)
    |   movel(pose_trans(ref_frame,p[0.099361, 0.081963, -0.000125, -0.013708, 3.141563, 0.000000]),accel_mss,speed_ms,0,0.001)
    |   movel(pose_trans(ref_frame,p[0.099104, 0.082297, -0.000125, -0.013708, 3.141563, 0.000000]),accel_mss,speed_ms,0,0.001)
    |   movel(pose_trans(ref_frame,p[0.098795, 0.082577, -0.000125, -0.013708, 3.141563, 0.000000]),accel_mss,speed_ms,0,0.001)
    |   movel(pose_trans(ref_frame,p[0.098440, 0.082796, -0.000125, -0.013708, 3.141563, 0.000000]),accel_mss,speed_ms,0,0.001)
    |   movel(pose_trans(ref_frame,p[0.098056, 0.082945, -0.000125, -0.013708, 3.141563, -0.000000]),accel_mss,speed_ms,0,0.001)
    |   movel(pose_trans(ref_frame,p[0.097650, 0.083020, -0.000125, -0.013708, 3.141563, 0.000000]),accel_mss,speed_ms,0,0.001)
    |   movel(pose_trans(ref_frame,p[0.097240, 0.083019, -0.000125, -0.013708, 3.141563, 0.000000]),accel_mss,speed_ms,0,0.001)
    |   movel(pose_trans(ref_frame,p[0.096838, 0.082941, -0.000125, -0.013708, 3.141563, 0.000000]),accel_mss,speed_ms,0,0.001)
    |   movel(pose_trans(ref_frame,p[0.096576, 0.082851, -0.000125, -0.013708, 3.141563, -0.000000]),accel_mss,speed_ms,0,0.001)
    |   movel(pose_trans(ref_frame,p[0.096324, 0.082738, -0.000125, -0.013708, 3.141563, -0.000000]),accel_mss,speed_ms,0,0.001)
    |   movel(pose_trans(ref_frame,p[0.096109, 0.082613, -0.000125, -0.013708, 3.141563, 0.000000]),accel_mss,speed_ms,0,0.001)
    |   movel(pose_trans(ref_frame,p[0.095911, 0.082463, -0.000125, -0.013708, 3.141563, -0.000000]),accel_mss,speed_ms,0,0.001)
    |   movel(pose_trans(ref_frame,p[0.095738, 0.082295, -0.000125, -0.013708, 3.141563, 0.000000]),accel_mss,speed_ms,0,0.001)
    |   movel(pose_trans(ref_frame,p[0.095588, 0.082105, -0.000125, -0.013708, 3.141563, -0.000000]),accel_mss,speed_ms,0,0.001)
    |   movel(pose_trans(ref_frame,p[0.095454, 0.081888, -0.000125, -0.013708, 3.141563, 0.000000]),accel_mss,speed_ms,0,0.001)
    |   movel(pose_trans(ref_frame,p[0.095344, 0.081657, -0.000125, -0.013708, 3.141563, 0.000000]),accel_mss,speed_ms,0,0.001)
    |   movel(pose_trans(ref_frame,p[0.095284, 0.081467, -0.000125, -0.013708, 3.141563, -0.000000]),accel_mss,speed_ms,0,0.001)
    |   movel(pose_trans(ref_frame,p[0.095257, 0.081269, -0.000125, -0.013708, 3.141563, 0.000000]),accel_mss,speed_ms,0,0.001)
    |   movel(pose_trans(ref_frame,p[0.095227, 0.080615, -0.000125, -0.013708, 3.141563, -0.000000]),accel_mss,speed_ms,0,0.001)
    |   movel(pose_trans(ref_frame,p[0.095203, 0.079961, -0.000125, -0.013708, 3.141563, 0.000000]),accel_mss,speed_ms,0,0.001)
    |   movel(pose_trans(ref_frame,p[0.095179, 0.079079, -0.000125, -0.013708, 3.141563, 0.000000]),accel_mss,speed_ms,0,0.001)
    |   movel(pose_trans(ref_frame,p[0.095165, 0.078196, -0.000125, -0.013708, 3.141563, 0.000000]),accel_mss,speed_ms,0,0.001)
    |   movel(pose_trans(ref_frame,p[0.095156, 0.076976, -0.000125, -0.013708, 3.141563, 0.000000]),accel_mss,speed_ms,0,0.001)
    |   movel(pose_trans(ref_frame,p[0.095152, 0.075756, -0.000125, -0.013708, 3.141563, 0.000000]),accel_mss,speed_ms,0,0.001)
    |   movel(pose_trans(ref_frame,p[0.095145, 0.070303, -0.000125, -0.013708, 3.141563, 0.000000]),accel_mss,speed_ms,0,0.001)
    |   movel(pose_trans(ref_frame,p[0.094424, 0.069924, -0.000125, -0.013708, 3.141563, 0.000000]),accel_mss,speed_ms,0,0.001)
    |   movel(pose_trans(ref_frame,p[0.094083, 0.069735, -0.000125, -0.013708, 3.141563, -0.000000]),accel_mss,speed_ms,0,0.001)
    |   movel(pose_trans(ref_frame,p[0.093753, 0.069530, -0.000125, -0.013708, 3.141563, 0.000000]),accel_mss,speed_ms,0,0.001)
    |   movel(pose_trans(ref_frame,p[0.093454, 0.069324, -0.000125, -0.013708, 3.141563, 0.000000]),accel_mss,speed_ms,0,0.001)
    |   movel(pose_trans(ref_frame,p[0.093169, 0.069100, -0.000125, -0.013708, 3.141563, 0.000000]),accel_mss,speed_ms,0,0.001)
    |   movel(pose_trans(ref_frame,p[0.092915, 0.068876, -0.000125, -0.013708, 3.141563, -0.000000]),accel_mss,speed_ms,0,0.001)
    |   movel(pose_trans(ref_frame,p[0.092676, 0.068636, -0.000125, -0.013708, 3.141563, 0.000000]),accel_mss,speed_ms,0,0.001)
    |   movel(pose_trans(ref_frame,p[0.092468, 0.068396, -0.000125, -0.013708, 3.141563, 0.000000]),accel_mss,speed_ms,0,0.001)
    |   movel(pose_trans(ref_frame,p[0.092278, 0.068141, -0.000125, -0.013708, 3.141563, -0.000000]),accel_mss,speed_ms,0,0.001)
    |   movel(pose_trans(ref_frame,p[0.092147, 0.067962, -0.000125, -0.013708, 3.141563, -0.000000]),accel_mss,speed_ms,0,0.001)
    |   movel(pose_trans(ref_frame,p[0.092008, 0.067790, -0.000125, -0.013708, 3.141563, -0.000000]),accel_mss,speed_ms,0,0.001)
    |   movel(pose_trans(ref_frame,p[0.091902, 0.067687, -0.000125, -0.013708, 3.141563, 0.000000]),accel_mss,speed_ms,0,0.001)
    |   movel(pose_trans(ref_frame,p[0.091781, 0.067602, -0.000125, -0.013708, 3.141563, 0.000000]),accel_mss,speed_ms,0,0.001)
    |   movel(pose_trans(ref_frame,p[0.091687, 0.067566, -0.000125, -0.013708, 3.141563, 0.000000]),accel_mss,speed_ms,0,0.001)
    |   movel(pose_trans(ref_frame,p[0.091586, 0.067560, -0.000125, -0.013708, 3.141563, -0.000000]),accel_mss,speed_ms,0,0.001)
    |   movel(pose_trans(ref_frame,p[0.091492, 0.067586, -0.000125, -0.013708, 3.141563, 0.000000]),accel_mss,speed_ms,0,0.001)
    |   movel(pose_trans(ref_frame,p[0.091412, 0.067642, -0.000125, -0.013708, 3.141563, -0.000000]),accel_mss,speed_ms,0,0.001)
    |   movel(pose_trans(ref_frame,p[0.091335, 0.067757, -0.000125, -0.013708, 3.141563, -0.000000]),accel_mss,speed_ms,0,0.001)
    |   movel(pose_trans(ref_frame,p[0.091308, 0.067892, -0.000125, -0.013708, 3.141563, 0.000000]),accel_mss,speed_ms,0,0.001)
    |   movel(pose_trans(ref_frame,p[0.091309, 0.074338, -0.000125, -0.013708, 3.141563, 0.000000]),accel_mss,speed_ms,0,0.001)
    |   movel(pose_trans(ref_frame,p[0.091312, 0.077347, -0.000125, -0.013708, 3.141563, 0.000000]),accel_mss,speed_ms,0,0.001)
    |   movel(pose_trans(ref_frame,p[0.091322, 0.080356, -0.000125, -0.013708, 3.141563, -0.000000]),accel_mss,speed_ms,0,0.001)
    |   movel(pose_trans(ref_frame,p[0.091347, 0.081015, -0.000125, -0.013708, 3.141563, 0.000000]),accel_mss,speed_ms,0,0.001)
    |   movel(pose_trans(ref_frame,p[0.091418, 0.081670, -0.000125, -0.013708, 3.141563, -0.000000]),accel_mss,speed_ms,0,0.001)
    |   movel(pose_trans(ref_frame,p[0.091504, 0.082134, -0.000125, -0.013708, 3.141563, 0.000000]),accel_mss,speed_ms,0,0.001)
    |   movel(pose_trans(ref_frame,p[0.091627, 0.082590, -0.000125, -0.013708, 3.141563, 0.000000]),accel_mss,speed_ms,0,0.001)
    |   movel(pose_trans(ref_frame,p[0.091791, 0.083050, -0.000125, -0.013708, 3.141563, 0.000000]),accel_mss,speed_ms,0,0.001)
    |   movel(pose_trans(ref_frame,p[0.091987, 0.083496, -0.000125, -0.013708, 3.141563, 0.000000]),accel_mss,speed_ms,0,0.001)
    |   movel(pose_trans(ref_frame,p[0.092217, 0.083929, -0.000125, -0.013708, 3.141563, 0.000000]),accel_mss,speed_ms,0,0.001)
    |   movel(pose_trans(ref_frame,p[0.092477, 0.084343, -0.000125, -0.013708, 3.141563, 0.000000]),accel_mss,speed_ms,0,0.001)
    |   movel(pose_trans(ref_frame,p[0.092760, 0.084726, -0.000125, -0.013708, 3.141563, 0.000000]),accel_mss,speed_ms,0,0.001)
    |   movel(pose_trans(ref_frame,p[0.093073, 0.085084, -0.000125, -0.013708, 3.141563, -0.000000]),accel_mss,speed_ms,0,0.001)
    |   movel(pose_trans(ref_frame,p[0.093151, 0.085162, -0.000125, -0.013708, 3.141563, 0.000000]),accel_mss,speed_ms,0,0.001)
    |   movel(pose_trans(ref_frame,p[0.093233, 0.085234, -0.000125, -0.013708, 3.141563, 0.000000]),accel_mss,speed_ms,0,0.001)
    |   movel(pose_trans(ref_frame,p[0.093361, 0.085338, -0.000125, -0.013708, 3.141563, -0.000000]),accel_mss,speed_ms,0,0.001)
    |   movel(pose_trans(ref_frame,p[0.093490, 0.085440, -0.000125, -0.013708, 3.141563, 0.000000]),accel_mss,speed_ms,0,0.001)
    |   movel(pose_trans(ref_frame,p[0.093638, 0.085551, -0.000125, -0.013708, 3.141563, 0.000000]),accel_mss,speed_ms,0,0.001)
    |   movel(pose_trans(ref_frame,p[0.093788, 0.085660, -0.000125, -0.013708, 3.141563, -0.000000]),accel_mss,speed_ms,0,0.001)
    |   movel(pose_trans(ref_frame,p[0.093936, 0.085763, -0.000125, -0.013708, 3.141563, 0.000000]),accel_mss,speed_ms,0,0.001)
    |   movel(pose_trans(ref_frame,p[0.094086, 0.085863, -0.000125, -0.013708, 3.141563, -0.000000]),accel_mss,speed_ms,0,0) # end trace
    |   speed_ms    = 1.000
    |   movel(pose_trans(ref_frame,p[0.094089, 0.085862, 0.005000, -0.013708, 3.141563, 0.000000]),accel_mss,speed_ms,0,0.001)
    |   movel(pose_trans(ref_frame,p[0.108316, 0.086915, 0.005000, -0.013708, 3.141563, -0.000000]),accel_mss,speed_ms,0,0) # end trace
    |   speed_ms    = 0.002
    |   movel(pose_trans(ref_frame,p[0.108316, 0.086915, -0.000125, -0.013708, 3.141563, -0.000000]),accel_mss,speed_ms,0,0) # end trace
    |   speed_ms    = 0.007
    |   movel(pose_trans(ref_frame,p[0.109637, 0.086909, -0.000125, -0.013708, 3.141563, 0.000000]),accel_mss,speed_ms,0,0.001)
    |   movel(pose_trans(ref_frame,p[0.110957, 0.086897, -0.000125, -0.013708, 3.141563, 0.000000]),accel_mss,speed_ms,0,0.001)
    |   movel(pose_trans(ref_frame,p[0.112125, 0.086882, -0.000125, -0.013708, 3.141563, -0.000000]),accel_mss,speed_ms,0,0.001)
    |   movel(pose_trans(ref_frame,p[0.113294, 0.086859, -0.000125, -0.013708, 3.141563, 0.000000]),accel_mss,speed_ms,0,0.001)
    |   movel(pose_trans(ref_frame,p[0.114283, 0.086835, -0.000125, -0.013708, 3.141563, 0.000000]),accel_mss,speed_ms,0,0.001)
    |   movel(pose_trans(ref_frame,p[0.115271, 0.086809, -0.000125, -0.013708, 3.141563, 0.000000]),accel_mss,speed_ms,0,0.001)
    |   movel(pose_trans(ref_frame,p[0.115520, 0.086791, -0.000125, -0.013708, 3.141563, 0.000000]),accel_mss,speed_ms,0,0.001)
    |   movel(pose_trans(ref_frame,p[0.115766, 0.086750, -0.000125, -0.013708, 3.141563, 0.000000]),accel_mss,speed_ms,0,0.001)
    |   movel(pose_trans(ref_frame,p[0.116154, 0.086655, -0.000125, -0.013708, 3.141563, 0.000000]),accel_mss,speed_ms,0,0.001)
    |   movel(pose_trans(ref_frame,p[0.116535, 0.086536, -0.000125, -0.013708, 3.141563, 0.000000]),accel_mss,speed_ms,0,0.001)
    |   movel(pose_trans(ref_frame,p[0.116891, 0.086399, -0.000125, -0.013708, 3.141563, 0.000000]),accel_mss,speed_ms,0,0.001)
    |   movel(pose_trans(ref_frame,p[0.117235, 0.086238, -0.000125, -0.013708, 3.141563, -0.000000]),accel_mss,speed_ms,0,0.001)
    |   movel(pose_trans(ref_frame,p[0.117572, 0.086051, -0.000125, -0.013708, 3.141563, 0.000000]),accel_mss,speed_ms,0,0.001)
    |   movel(pose_trans(ref_frame,p[0.117895, 0.085840, -0.000125, -0.013708, 3.141563, 0.000000]),accel_mss,speed_ms,0,0.001)
    |   movel(pose_trans(ref_frame,p[0.118226, 0.085594, -0.000125, -0.013708, 3.141563, -0.000000]),accel_mss,speed_ms,0,0.001)
    |   movel(pose_trans(ref_frame,p[0.118542, 0.085329, -0.000125, -0.013708, 3.141563, 0.000000]),accel_mss,speed_ms,0,0.001)
    |   movel(pose_trans(ref_frame,p[0.119190, 0.084667, -0.000125, -0.013708, 3.141563, -0.000000]),accel_mss,speed_ms,0,0.001)
    |   movel(pose_trans(ref_frame,p[0.119738, 0.083919, -0.000125, -0.013708, 3.141563, 0.000000]),accel_mss,speed_ms,0,0.001)
    |   movel(pose_trans(ref_frame,p[0.120156, 0.083124, -0.000125, -0.013708, 3.141563, 0.000000]),accel_mss,speed_ms,0,0.001)
    |   movel(pose_trans(ref_frame,p[0.120445, 0.082273, -0.000125, -0.013708, 3.141563, -0.000000]),accel_mss,speed_ms,0,0.001)
    |   movel(pose_trans(ref_frame,p[0.120600, 0.081385, -0.000125, -0.013708, 3.141563, -0.000000]),accel_mss,speed_ms,0,0.001)
    |   movel(pose_trans(ref_frame,p[0.120615, 0.080483, -0.000125, -0.013708, 3.141563, -0.000000]),accel_mss,speed_ms,0,0.001)
    |   movel(pose_trans(ref_frame,p[0.120494, 0.079556, -0.000125, -0.013708, 3.141563, -0.000000]),accel_mss,speed_ms,0,0.001)
    |   movel(pose_trans(ref_frame,p[0.120246, 0.078653, -0.000125, -0.013708, 3.141563, 0.000000]),accel_mss,speed_ms,0,0.001)
    |   movel(pose_trans(ref_frame,p[0.120132, 0.078341, -0.000125, -0.013708, 3.141563, 0.000000]),accel_mss,speed_ms,0,0.001)
    |   movel(pose_trans(ref_frame,p[0.120011, 0.078032, -0.000125, -0.013708, 3.141563, -0.000000]),accel_mss,speed_ms,0,0.001)
    |   movel(pose_trans(ref_frame,p[0.119917, 0.077822, -0.000125, -0.013708, 3.141563, 0.000000]),accel_mss,speed_ms,0,0.001)
    |   movel(pose_trans(ref_frame,p[0.119809, 0.077620, -0.000125, -0.013708, 3.141563, 0.000000]),accel_mss,speed_ms,0,0.001)
    |   movel(pose_trans(ref_frame,p[0.119690, 0.077431, -0.000125, -0.013708, 3.141563, 0.000000]),accel_mss,speed_ms,0,0.001)
    |   movel(pose_trans(ref_frame,p[0.119558, 0.077252, -0.000125, -0.013708, 3.141563, -0.000000]),accel_mss,speed_ms,0,0.001)
    |   movel(pose_trans(ref_frame,p[0.119363, 0.077013, -0.000125, -0.013708, 3.141563, 0.000000]),accel_mss,speed_ms,0,0.001)
    |   movel(pose_trans(ref_frame,p[0.119161, 0.076781, -0.000125, -0.013708, 3.141563, -0.000000]),accel_mss,speed_ms,0,0.001)
    |   movel(pose_trans(ref_frame,p[0.118639, 0.076247, -0.000125, -0.013708, 3.141563, 0.000000]),accel_mss,speed_ms,0,0.001)
    |   movel(pose_trans(ref_frame,p[0.118071, 0.075764, -0.000125, -0.013708, 3.141563, 0.000000]),accel_mss,speed_ms,0,0.001)
    |   movel(pose_trans(ref_frame,p[0.117528, 0.075399, -0.000125, -0.013708, 3.141563, -0.000000]),accel_mss,speed_ms,0,0.001)
    |   movel(pose_trans(ref_frame,p[0.116940, 0.075112, -0.000125, -0.013708, 3.141563, -0.000000]),accel_mss,speed_ms,0,0.001)
    |   movel(pose_trans(ref_frame,p[0.116284, 0.074891, -0.000125, -0.013708, 3.141563, 0.000000]),accel_mss,speed_ms,0,0.001)
    |   movel(pose_trans(ref_frame,p[0.115605, 0.074754, -0.000125, -0.013708, 3.141563, -0.000000]),accel_mss,speed_ms,0,0.001)
    |   movel(pose_trans(ref_frame,p[0.114746, 0.074663, -0.000125, -0.013708, 3.141563, -0.000000]),accel_mss,speed_ms,0,0.001)
    |   movel(pose_trans(ref_frame,p[0.113883, 0.074629, -0.000125, -0.013708, 3.141563, 0.000000]),accel_mss,speed_ms,0,0.001)
    |   movel(pose_trans(ref_frame,p[0.112221, 0.074617, -0.000125, -0.013708, 3.141563, 0.000000]),accel_mss,speed_ms,0,0.001)
    |   movel(pose_trans(ref_frame,p[0.112215, 0.072755, -0.000125, -0.013708, 3.141563, 0.000000]),accel_mss,speed_ms,0,0.001)
    |   movel(pose_trans(ref_frame,p[0.112213, 0.072394, -0.000125, -0.013708, 3.141563, -0.000000]),accel_mss,speed_ms,0,0.001)
    |   movel(pose_trans(ref_frame,p[0.112208, 0.072034, -0.000125, -0.013708, 3.141563, -0.000000]),accel_mss,speed_ms,0,0.001)
    |   movel(pose_trans(ref_frame,p[0.112202, 0.071720, -0.000125, -0.013708, 3.141563, 0.000000]),accel_mss,speed_ms,0,0.001)
    |   movel(pose_trans(ref_frame,p[0.112194, 0.071406, -0.000125, -0.013708, 3.141563, 0.000000]),accel_mss,speed_ms,0,0.001)
    |   movel(pose_trans(ref_frame,p[0.112184, 0.071138, -0.000125, -0.013708, 3.141563, 0.000000]),accel_mss,speed_ms,0,0.001)
    |   movel(pose_trans(ref_frame,p[0.112174, 0.070869, -0.000125, -0.013708, 3.141563, -0.000000]),accel_mss,speed_ms,0,0.001)
    |   movel(pose_trans(ref_frame,p[0.112168, 0.070821, -0.000125, -0.013708, 3.141563, -0.000000]),accel_mss,speed_ms,0,0.001)
    |   movel(pose_trans(ref_frame,p[0.112151, 0.070776, -0.000125, -0.013708, 3.141563, -0.000000]),accel_mss,speed_ms,0,0.001)
    |   movel(pose_trans(ref_frame,p[0.112092, 0.070711, -0.000125, -0.013708, 3.141563, 0.000000]),accel_mss,speed_ms,0,0.001)
    |   movel(pose_trans(ref_frame,p[0.112008, 0.070685, -0.000125, -0.013708, 3.141563, -0.000000]),accel_mss,speed_ms,0,0.001)
    |   movel(pose_trans(ref_frame,p[0.111602, 0.070675, -0.000125, -0.013708, 3.141563, -0.000000]),accel_mss,speed_ms,0,0.001)
    |   movel(pose_trans(ref_frame,p[0.111196, 0.070665, -0.000125, -0.013708, 3.141563, 0.000000]),accel_mss,speed_ms,0,0.001)
    |   movel(pose_trans(ref_frame,p[0.110767, 0.070656, -0.000125, -0.013708, 3.141563, 0.000000]),accel_mss,speed_ms,0,0.001)
    |   movel(pose_trans(ref_frame,p[0.110339, 0.070647, -0.000125, -0.013708, 3.141563, -0.000000]),accel_mss,speed_ms,0,0.001)
    |   movel(pose_trans(ref_frame,p[0.109945, 0.070639, -0.000125, -0.013708, 3.141563, 0.000000]),accel_mss,speed_ms,0,0.001)
    |   movel(pose_trans(ref_frame,p[0.109551, 0.070632, -0.000125, -0.013708, 3.141563, -0.000000]),accel_mss,speed_ms,0,0.001)
    |   movel(pose_trans(ref_frame,p[0.109118, 0.070625, -0.000125, -0.013708, 3.141563, 0.000000]),accel_mss,speed_ms,0,0.001)
    |   movel(pose_trans(ref_frame,p[0.108686, 0.070619, -0.000125, -0.013708, 3.141563, 0.000000]),accel_mss,speed_ms,0,0.001)
    |   movel(pose_trans(ref_frame,p[0.108576, 0.070640, -0.000125, -0.013708, 3.141563, 0.000000]),accel_mss,speed_ms,0,0.001)
    |   movel(pose_trans(ref_frame,p[0.108482, 0.070702, -0.000125, -0.013708, 3.141563, -0.000000]),accel_mss,speed_ms,0,0.001)
    |   movel(pose_trans(ref_frame,p[0.108407, 0.070815, -0.000125, -0.013708, 3.141563, 0.000000]),accel_mss,speed_ms,0,0.001)
    |   movel(pose_trans(ref_frame,p[0.108380, 0.070948, -0.000125, -0.013708, 3.141563, -0.000000]),accel_mss,speed_ms,0,0.001)
    |   movel(pose_trans(ref_frame,p[0.108392, 0.076497, -0.000125, -0.013708, 3.141563, 0.000000]),accel_mss,speed_ms,0,0.001)
    |   movel(pose_trans(ref_frame,p[0.108409, 0.082045, -0.000125, -0.013708, 3.141563, 0.000000]),accel_mss,speed_ms,0,0.001)
    |   movel(pose_trans(ref_frame,p[0.108436, 0.082179, -0.000125, -0.013708, 3.141563, -0.000000]),accel_mss,speed_ms,0,0.001)
    |   movel(pose_trans(ref_frame,p[0.108512, 0.082292, -0.000125, -0.013708, 3.141563, -0.000000]),accel_mss,speed_ms,0,0.001)
    |   movel(pose_trans(ref_frame,p[0.108646, 0.082383, -0.000125, -0.013708, 3.141563, -0.000000]),accel_mss,speed_ms,0,0.001)
    |   movel(pose_trans(ref_frame,p[0.108805, 0.082417, -0.000125, -0.013708, 3.141563, 0.000000]),accel_mss,speed_ms,0,0.001)
    |   movel(pose_trans(ref_frame,p[0.109547, 0.082429, -0.000125, -0.013708, 3.141563, 0.000000]),accel_mss,speed_ms,0,0.001)
    |   movel(pose_trans(ref_frame,p[0.110290, 0.082434, -0.000125, -0.013708, 3.141563, 0.000000]),accel_mss,speed_ms,0,0.001)
    |   movel(pose_trans(ref_frame,p[0.111032, 0.082431, -0.000125, -0.013708, 3.141563, -0.000000]),accel_mss,speed_ms,0,0.001)
    |   movel(pose_trans(ref_frame,p[0.111775, 0.082422, -0.000125, -0.013708, 3.141563, -0.000000]),accel_mss,speed_ms,0,0.001)
    |   movel(pose_trans(ref_frame,p[0.111933, 0.082388, -0.000125, -0.013708, 3.141563, -0.000000]),accel_mss,speed_ms,0,0.001)
    |   movel(pose_trans(ref_frame,p[0.112067, 0.082298, -0.000125, -0.013708, 3.141563, 0.000000]),accel_mss,speed_ms,0,0.001)
    |   movel(pose_trans(ref_frame,p[0.112106, 0.082243, -0.000125, -0.013708, 3.141563, 0.000000]),accel_mss,speed_ms,0,0.001)
    |   movel(pose_trans(ref_frame,p[0.112123, 0.082178, -0.000125, -0.013708, 3.141563, 0.000000]),accel_mss,speed_ms,0,0.001)
    |   movel(pose_trans(ref_frame,p[0.112147, 0.081919, -0.000125, -0.013708, 3.141563, 0.000000]),accel_mss,speed_ms,0,0.001)
    |   movel(pose_trans(ref_frame,p[0.112168, 0.081659, -0.000125, -0.013708, 3.141563, 0.000000]),accel_mss,speed_ms,0,0.001)
    |   movel(pose_trans(ref_frame,p[0.112187, 0.081348, -0.000125, -0.013708, 3.141563, 0.000000]),accel_mss,speed_ms,0,0.001)
    |   movel(pose_trans(ref_frame,p[0.112200, 0.081036, -0.000125, -0.013708, 3.141563, 0.000000]),accel_mss,speed_ms,0,0.001)
    |   movel(pose_trans(ref_frame,p[0.112208, 0.080680, -0.000125, -0.013708, 3.141563, 0.000000]),accel_mss,speed_ms,0,0.001)
    |   movel(pose_trans(ref_frame,p[0.112211, 0.080323, -0.000125, -0.013708, 3.141563, 0.000000]),accel_mss,speed_ms,0,0.001)
    |   movel(pose_trans(ref_frame,p[0.112214, 0.078490, -0.000125, -0.013708, 3.141563, 0.000000]),accel_mss,speed_ms,0,0.001)
    |   movel(pose_trans(ref_frame,p[0.113576, 0.078486, -0.000125, -0.013708, 3.141563, 0.000000]),accel_mss,speed_ms,0,0.001)
    |   movel(pose_trans(ref_frame,p[0.114102, 0.078496, -0.000125, -0.013708, 3.141563, 0.000000]),accel_mss,speed_ms,0,0.001)
    |   movel(pose_trans(ref_frame,p[0.114628, 0.078527, -0.000125, -0.013708, 3.141563, -0.000000]),accel_mss,speed_ms,0,0.001)
    |   movel(pose_trans(ref_frame,p[0.114985, 0.078578, -0.000125, -0.013708, 3.141563, 0.000000]),accel_mss,speed_ms,0,0.001)
    |   movel(pose_trans(ref_frame,p[0.115332, 0.078673, -0.000125, -0.013708, 3.141563, -0.000000]),accel_mss,speed_ms,0,0.001)
    |   movel(pose_trans(ref_frame,p[0.115609, 0.078794, -0.000125, -0.013708, 3.141563, -0.000000]),accel_mss,speed_ms,0,0.001)
    |   movel(pose_trans(ref_frame,p[0.115862, 0.078958, -0.000125, -0.013708, 3.141563, -0.000000]),accel_mss,speed_ms,0,0.001)
    |   movel(pose_trans(ref_frame,p[0.116113, 0.079178, -0.000125, -0.013708, 3.141563, -0.000000]),accel_mss,speed_ms,0,0.001)
    |   movel(pose_trans(ref_frame,p[0.116335, 0.079427, -0.000125, -0.013708, 3.141563, 0.000000]),accel_mss,speed_ms,0,0.001)
    |   movel(pose_trans(ref_frame,p[0.116488, 0.079647, -0.000125, -0.013708, 3.141563, 0.000000]),accel_mss,speed_ms,0,0.001)
    |   movel(pose_trans(ref_frame,p[0.116613, 0.079885, -0.000125, -0.013708, 3.141563, 0.000000]),accel_mss,speed_ms,0,0.001)
    |   movel(pose_trans(ref_frame,p[0.116708, 0.080137, -0.000125, -0.013708, 3.141563, 0.000000]),accel_mss,speed_ms,0,0.001)
    |   movel(pose_trans(ref_frame,p[0.116772, 0.080399, -0.000125, -0.013708, 3.141563, 0.000000]),accel_mss,speed_ms,0,0.001)
    |   movel(pose_trans(ref_frame,p[0.116804, 0.080665, -0.000125, -0.013708, 3.141563, 0.000000]),accel_mss,speed_ms,0,0.001)
    |   movel(pose_trans(ref_frame,p[0.116803, 0.080934, -0.000125, -0.013708, 3.141563, 0.000000]),accel_mss,speed_ms,0,0.001)
    |   movel(pose_trans(ref_frame,p[0.116770, 0.081198, -0.000125, -0.013708, 3.141563, 0.000000]),accel_mss,speed_ms,0,0.001)
    |   movel(pose_trans(ref_frame,p[0.116704, 0.081456, -0.000125, -0.013708, 3.141563, -0.000000]),accel_mss,speed_ms,0,0.001)
    |   movel(pose_trans(ref_frame,p[0.116620, 0.081661, -0.000125, -0.013708, 3.141563, -0.000000]),accel_mss,speed_ms,0,0.001)
    |   movel(pose_trans(ref_frame,p[0.116508, 0.081851, -0.000125, -0.013708, 3.141563, 0.000000]),accel_mss,speed_ms,0,0.001)
    |   movel(pose_trans(ref_frame,p[0.116339, 0.082079, -0.000125, -0.013708, 3.141563, -0.000000]),accel_mss,speed_ms,0,0.001)
    |   movel(pose_trans(ref_frame,p[0.116154, 0.082295, -0.000125, -0.013708, 3.141563, 0.000000]),accel_mss,speed_ms,0,0.001)
    |   movel(pose_trans(ref_frame,p[0.115952, 0.082499, -0.000125, -0.013708, 3.141563, 0.000000]),accel_mss,speed_ms,0,0.001)
    |   movel(pose_trans(ref_frame,p[0.115737, 0.082688, -0.000125, -0.013708, 3.141563, -0.000000]),accel_mss,speed_ms,0,0.001)
    |   movel(pose_trans(ref_frame,p[0.115549, 0.082823, -0.000125, -0.013708, 3.141563, 0.000000]),accel_mss,speed_ms,0,0.001)
    |   movel(pose_trans(ref_frame,p[0.115345, 0.082931, -0.000125, -0.013708, 3.141563, -0.000000]),accel_mss,speed_ms,0,0.001)
    |   movel(pose_trans(ref_frame,p[0.115218, 0.082974, -0.000125, -0.013708, 3.141563, 0.000000]),accel_mss,speed_ms,0,0.001)
    |   movel(pose_trans(ref_frame,p[0.115085, 0.082991, -0.000125, -0.013708, 3.141563, -0.000000]),accel_mss,speed_ms,0,0.001)
    |   movel(pose_trans(ref_frame,p[0.114293, 0.083016, -0.000125, -0.013708, 3.141563, -0.000000]),accel_mss,speed_ms,0,0.001)
    |   movel(pose_trans(ref_frame,p[0.113500, 0.083039, -0.000125, -0.013708, 3.141563, 0.000000]),accel_mss,speed_ms,0,0.001)
    |   movel(pose_trans(ref_frame,p[0.112578, 0.083060, -0.000125, -0.013708, 3.141563, -0.000000]),accel_mss,speed_ms,0,0.001)
    |   movel(pose_trans(ref_frame,p[0.111656, 0.083075, -0.000125, -0.013708, 3.141563, 0.000000]),accel_mss,speed_ms,0,0.001)
    |   movel(pose_trans(ref_frame,p[0.110593, 0.083084, -0.000125, -0.013708, 3.141563, 0.000000]),accel_mss,speed_ms,0,0.001)
    |   movel(pose_trans(ref_frame,p[0.109530, 0.083089, -0.000125, -0.013708, 3.141563, -0.000000]),accel_mss,speed_ms,0,0.001)
    |   movel(pose_trans(ref_frame,p[0.104046, 0.083098, -0.000125, -0.013708, 3.141563, -0.000000]),accel_mss,speed_ms,0,0.001)
    |   movel(pose_trans(ref_frame,p[0.103753, 0.083708, -0.000125, -0.013708, 3.141563, 0.000000]),accel_mss,speed_ms,0,0.001)
    |   movel(pose_trans(ref_frame,p[0.103661, 0.083885, -0.000125, -0.013708, 3.141563, 0.000000]),accel_mss,speed_ms,0,0.001)
    |   movel(pose_trans(ref_frame,p[0.103557, 0.084055, -0.000125, -0.013708, 3.141563, 0.000000]),accel_mss,speed_ms,0,0.001)
    |   movel(pose_trans(ref_frame,p[0.103428, 0.084243, -0.000125, -0.013708, 3.141563, 0.000000]),accel_mss,speed_ms,0,0.001)
    |   movel(pose_trans(ref_frame,p[0.103290, 0.084425, -0.000125, -0.013708, 3.141563, -0.000000]),accel_mss,speed_ms,0,0.001)
    |   movel(pose_trans(ref_frame,p[0.103111, 0.084644, -0.000125, -0.013708, 3.141563, -0.000000]),accel_mss,speed_ms,0,0.001)
    |   movel(pose_trans(ref_frame,p[0.102924, 0.084856, -0.000125, -0.013708, 3.141563, 0.000000]),accel_mss,speed_ms,0,0.001)
    |   movel(pose_trans(ref_frame,p[0.102670, 0.085131, -0.000125, -0.013708, 3.141563, 0.000000]),accel_mss,speed_ms,0,0.001)
    |   movel(pose_trans(ref_frame,p[0.102412, 0.085403, -0.000125, -0.013708, 3.141563, 0.000000]),accel_mss,speed_ms,0,0.001)
    |   movel(pose_trans(ref_frame,p[0.102209, 0.085613, -0.000125, -0.013708, 3.141563, 0.000000]),accel_mss,speed_ms,0,0.001)
    |   movel(pose_trans(ref_frame,p[0.102006, 0.085823, -0.000125, -0.013708, 3.141563, 0.000000]),accel_mss,speed_ms,0,0.001)
    |   movel(pose_trans(ref_frame,p[0.101830, 0.086006, -0.000125, -0.013708, 3.141563, 0.000000]),accel_mss,speed_ms,0,0.001)
    |   movel(pose_trans(ref_frame,p[0.101655, 0.086189, -0.000125, -0.013708, 3.141563, 0.000000]),accel_mss,speed_ms,0,0.001)
    |   movel(pose_trans(ref_frame,p[0.101353, 0.086506, -0.000125, -0.013708, 3.141563, 0.000000]),accel_mss,speed_ms,0,0.001)
    |   movel(pose_trans(ref_frame,p[0.101330, 0.086532, -0.000125, -0.013708, 3.141563, -0.000000]),accel_mss,speed_ms,0,0.001)
    |   movel(pose_trans(ref_frame,p[0.101308, 0.086559, -0.000125, -0.013708, 3.141563, 0.000000]),accel_mss,speed_ms,0,0.001)
    |   movel(pose_trans(ref_frame,p[0.101291, 0.086685, -0.000125, -0.013708, 3.141563, 0.000000]),accel_mss,speed_ms,0,0.001)
    |   movel(pose_trans(ref_frame,p[0.101392, 0.086762, -0.000125, -0.013708, 3.141563, -0.000000]),accel_mss,speed_ms,0,0.001)
    |   movel(pose_trans(ref_frame,p[0.101935, 0.086821, -0.000125, -0.013708, 3.141563, -0.000000]),accel_mss,speed_ms,0,0.001)
    |   movel(pose_trans(ref_frame,p[0.102480, 0.086859, -0.000125, -0.013708, 3.141563, 0.000000]),accel_mss,speed_ms,0,0.001)
    |   movel(pose_trans(ref_frame,p[0.103450, 0.086897, -0.000125, -0.013708, 3.141563, -0.000000]),accel_mss,speed_ms,0,0.001)
    |   movel(pose_trans(ref_frame,p[0.104420, 0.086912, -0.000125, -0.013708, 3.141563, 0.000000]),accel_mss,speed_ms,0,0.001)
    |   movel(pose_trans(ref_frame,p[0.106368, 0.086917, -0.000125, -0.013708, 3.141563, -0.000000]),accel_mss,speed_ms,0,0.001)
    |   movel(pose_trans(ref_frame,p[0.108316, 0.086915, -0.000125, -0.013708, 3.141563, -0.000000]),accel_mss,speed_ms,0,0) # end trace
    |   speed_ms    = 1.000
    |   movel(pose_trans(ref_frame,p[0.108316, 0.086915, 0.005000, -0.013708, 3.141563, -0.000000]),accel_mss,speed_ms,0,0.001)
    |   movel(pose_trans(ref_frame,p[0.110203, 0.069872, 0.005000, -0.013708, 3.141563, -0.000000]),accel_mss,speed_ms,0,0) # end trace
    |   speed_ms    = 0.002
    |   movel(pose_trans(ref_frame,p[0.110203, 0.069872, -0.000125, -0.013708, 3.141563, 0.000000]),accel_mss,speed_ms,0,0) # end trace
    |   speed_ms    = 0.007
    |   movel(pose_trans(ref_frame,p[0.110771, 0.069878, -0.000125, -0.013708, 3.141563, 0.000000]),accel_mss,speed_ms,0,0.001)
    |   movel(pose_trans(ref_frame,p[0.111339, 0.069870, -0.000125, -0.013708, 3.141563, 0.000000]),accel_mss,speed_ms,0,0.001)
    |   movel(pose_trans(ref_frame,p[0.111850, 0.069868, -0.000125, -0.013708, 3.141563, 0.000000]),accel_mss,speed_ms,0,0.001)
    |   movel(pose_trans(ref_frame,p[0.112361, 0.069865, -0.000125, -0.013708, 3.141563, -0.000000]),accel_mss,speed_ms,0,0.001)
    |   movel(pose_trans(ref_frame,p[0.113287, 0.069857, -0.000125, -0.013708, 3.141563, -0.000000]),accel_mss,speed_ms,0,0.001)
    |   movel(pose_trans(ref_frame,p[0.114213, 0.069843, -0.000125, -0.013708, 3.141563, -0.000000]),accel_mss,speed_ms,0,0.001)
    |   movel(pose_trans(ref_frame,p[0.115021, 0.069827, -0.000125, -0.013708, 3.141563, -0.000000]),accel_mss,speed_ms,0,0.001)
    |   movel(pose_trans(ref_frame,p[0.115829, 0.069811, -0.000125, -0.013708, 3.141563, 0.000000]),accel_mss,speed_ms,0,0.001)
    |   movel(pose_trans(ref_frame,p[0.115919, 0.069799, -0.000125, -0.013708, 3.141563, -0.000000]),accel_mss,speed_ms,0,0.001)
